LIN {X 0,Y 573.289,Z 87.196,A -85,B 0,C 180,E1 -2345.628,E2 -2345.628} C_VEL
LIN {X 0,Y 573.282,Z 87.197,A -85,B 0,C 180,E1 -2348.46,E2 -2348.46} C_VEL
LIN {X 0,Y 573.272,Z 87.197,A -85,B 0,C 180,E1 -2351.312,E2 -2351.312} C_VEL
LIN {X 0,Y 573.282,Z 87.196,A -85,B 0,C 180,E1 -2354.425,E2 -2354.425} C_VEL
LIN {X 0,Y 573.257,Z 87.199,A -85,B 0,C 180,E1 -2357.112,E2 -2357.112} C_VEL
LIN {X 0,Y 573.248,Z 87.201,A -85,B 0,C 180,E1 -2360.077,E2 -2360.077} C_VEL
LIN {X 0,Y 573.234,Z 87.203,A -85,B 0,C 180,E1 -2363.1,E2 -2363.1} C_VEL
LIN {X 0,Y 573.246,Z 87.199,A -85,B 0,C 180,E1 -2364.375,E2 -2364.375} C_VEL
LIN {X 0,Y 572.621,Z 87.279,A -85,B 0,C 180,E1 -2364.961,E2 -2364.961} C_VEL
LIN {X 0,Y 569.781,Z 87.64,A -85,B 0,C 180,E1 -2365.912,E2 -2365.912} C_VEL
LIN {X 0,Y 567.349,Z 87.946,A -85,B 0,C 180,E1 -2366.678,E2 -2366.678} C_VEL
LIN {X 0,Y 566.294,Z 88.074,A -85,B 0,C 180,E1 -2367.269,E2 -2367.269} C_VEL
LIN {X 0,Y 566.203,Z 88.082,A -85,B 0,C 180,E1 -2367.469,E2 -2367.469} C_VEL
LIN {X 0,Y 566.196,Z 88.08,A -85,B 0,C 180,E1 -2369.769,E2 -2369.769} C_VEL
LIN {X 0,Y 566.202,Z 88.076,A -85,B 0,C 180,E1 -2372.43,E2 -2372.43} C_VEL
LIN {X 0,Y 566.179,Z 88.086,A -85,B 0,C 180,E1 -2374.99,E2 -2374.99} C_VEL
LIN {X 0,Y 566.196,Z 88.08,A -85,B 0,C 180,E1 -2377.461,E2 -2377.461} C_VEL
LIN {X 0,Y 566.207,Z 88.076,A -85,B 0,C 180,E1 -2380.199,E2 -2380.199} C_VEL
LIN {X 0,Y 566.198,Z 88.083,A -85,B 0,C 180,E1 -2383.055,E2 -2383.055} C_VEL
LIN {X 0,Y 566.194,Z 88.078,A -85,B 0,C 180,E1 -2386.05,E2 -2386.05} C_VEL
LIN {X 0,Y 566.204,Z 88.078,A -85,B 0,C 180,E1 -2389.215,E2 -2389.215} C_VEL
LIN {X 0,Y 566.182,Z 88.078,A -85,B 0,C 180,E1 -2391.637,E2 -2391.637} C_VEL
LIN {X 0,Y 566.151,Z 88.089,A -85,B 0,C 180,E1 -2394.307,E2 -2394.307} C_VEL
LIN {X 0,Y 566.221,Z 88.076,A -85,B 0,C 180,E1 -2396.898,E2 -2396.898} C_VEL
LIN {X 0,Y 566.18,Z 88.079,A -85,B 0,C 180,E1 -2399.407,E2 -2399.407} C_VEL
LIN {X 0,Y 566.189,Z 88.081,A -85,B 0,C 180,E1 -2401.856,E2 -2401.856} C_VEL
LIN {X 0,Y 566.24,Z 88.071,A -85,B 0,C 180,E1 -2405.039,E2 -2405.039} C_VEL
LIN {X 0,Y 566.194,Z 88.086,A -85,B 0,C 180,E1 -2408.138,E2 -2408.138} C_VEL
LIN {X 0,Y 566.234,Z 88.075,A -85,B 0,C 180,E1 -2410.614,E2 -2410.614} C_VEL
LIN {X 0,Y 566.2,Z 88.087,A -85,B 0,C 180,E1 -2413.783,E2 -2413.783} C_VEL
LIN {X 0,Y 566.208,Z 88.167,A -85,B 0,C 180,E1 -2414.153,E2 -2414.153} C_VEL
LIN {X 0,Y 566.918,Z 92.77,A -85,B 0,C 180,E1 -2414.91,E2 -2414.91} C_VEL
LIN {X 0,Y 566.626,Z 111.554,A -85,B 0,C 180,E1 -2417.828,E2 -2417.828} C_VEL
LIN {X 0,Y 566.562,Z 119.682,A -85,B 0,C 180,E1 -2419.076,E2 -2419.076} C_VEL
LIN {X 0,Y 567.768,Z 127.51,A -85,B 0,C 180,E1 -2419.22,E2 -2419.22} C_VEL
LIN {X 0,Y 567.41,Z 256.467,A -85,B 0,C 180,E1 -2420.891,E2 -2420.891} C_VEL
LIN {X 0,Y 567.294,Z 270.884,A -85,B 0,C 180,E1 -2421.226,E2 -2421.226} C_VEL
LIN {X 0,Y 567.151,Z 285.238,A -85,B 0,C 180,E1 -2421.718,E2 -2421.718} C_VEL
LIN {X 0,Y 566.971,Z 298.855,A -85,B 0,C 180,E1 -2422.343,E2 -2422.343} C_VEL
LIN {X 0,Y 566.759,Z 311.074,A -85,B 0,C 180,E1 -2423.055,E2 -2423.055} C_VEL
LIN {X 0,Y 566.617,Z 323.455,A -85,B 0,C 180,E1 -2423.948,E2 -2423.948} C_VEL
LIN {X 0,Y 566.381,Z 333.622,A -85,B 0,C 180,E1 -2424.839,E2 -2424.839} C_VEL
LIN {X 0,Y 566.246,Z 343.77,A -85,B 0,C 180,E1 -2425.908,E2 -2425.908} C_VEL
LIN {X 0,Y 566.124,Z 352.189,A -85,B 0,C 180,E1 -2426.976,E2 -2426.976} C_VEL
LIN {X 0,Y 566.109,Z 360.261,A -85,B 0,C 180,E1 -2428.222,E2 -2428.222} C_VEL
LIN {X 0,Y 565.936,Z 365.957,A -85,B 0,C 180,E1 -2429.289,E2 -2429.289} C_VEL
LIN {X 0,Y 565.95,Z 370.617,A -85,B 0,C 180,E1 -2430.356,E2 -2430.356} C_VEL
LIN {X 0,Y 565.9,Z 375.469,A -85,B 0,C 180,E1 -2431.779,E2 -2431.779} C_VEL
LIN {X 0,Y 565.873,Z 378.126,A -85,B 0,C 180,E1 -2432.848,E2 -2432.848} C_VEL
LIN {X 0,Y 565.91,Z 380.449,A -85,B 0,C 180,E1 -2434.273,E2 -2434.273} C_VEL
LIN {X 0,Y 565.895,Z 381.431,A -85,B 0,C 180,E1 -2435.702,E2 -2435.702} C_VEL
LIN {X 0,Y 565.885,Z 381.084,A -85,B 0,C 180,E1 -2437.134,E2 -2437.134} C_VEL
LIN {X 0,Y 565.853,Z 379.389,A -85,B 0,C 180,E1 -2438.572,E2 -2438.572} C_VEL
LIN {X 0,Y 565.913,Z 376.297,A -85,B 0,C 180,E1 -2440.013,E2 -2440.013} C_VEL
LIN {X 0,Y 565.942,Z 371.702,A -85,B 0,C 180,E1 -2441.461,E2 -2441.461} C_VEL
LIN {X 0,Y 565.955,Z 367.124,A -85,B 0,C 180,E1 -2442.551,E2 -2442.551} C_VEL
LIN {X 0,Y 566.033,Z 360.492,A -85,B 0,C 180,E1 -2443.828,E2 -2443.828} C_VEL
LIN {X 0,Y 566.123,Z 352.208,A -85,B 0,C 180,E1 -2445.112,E2 -2445.112} C_VEL
LIN {X 0,Y 566.243,Z 343.476,A -85,B 0,C 180,E1 -2446.216,E2 -2446.216} C_VEL
LIN {X 0,Y 566.418,Z 332.825,A -85,B 0,C 180,E1 -2447.325,E2 -2447.325} C_VEL
LIN {X 0,Y 566.578,Z 322.04,A -85,B 0,C 180,E1 -2448.253,E2 -2448.253} C_VEL
LIN {X 0,Y 566.775,Z 310.231,A -85,B 0,C 180,E1 -2449.089,E2 -2449.089} C_VEL
LIN {X 0,Y 566.988,Z 297.689,A -85,B 0,C 180,E1 -2449.807,E2 -2449.807} C_VEL
LIN {X 0,Y 567.161,Z 284.65,A -85,B 0,C 180,E1 -2450.396,E2 -2450.396} C_VEL
LIN {X 0,Y 567.302,Z 270.052,A -85,B 0,C 180,E1 -2450.889,E2 -2450.889} C_VEL
LIN {X 0,Y 567.409,Z 255.45,A -85,B 0,C 180,E1 -2451.216,E2 -2451.216} C_VEL
LIN {X 0,Y 567.666,Z 125.494,A -85,B 0,C 180,E1 -2452.9,E2 -2452.9} C_VEL
LIN {X 0,Y 566.565,Z 119.617,A -85,B 0,C 180,E1 -2453.025,E2 -2453.025} C_VEL
LIN {X 0,Y 566.783,Z 100.873,A -85,B 0,C 180,E1 -2455.919,E2 -2455.919} C_VEL
LIN {X 0,Y 566.816,Z 92.019,A -85,B 0,C 180,E1 -2457.308,E2 -2457.308} C_VEL
LIN {X 0,Y 566.144,Z 88.093,A -85,B 0,C 180,E1 -2457.995,E2 -2457.995} C_VEL
LIN {X 0,Y 566.173,Z 88.082,A -85,B 0,C 180,E1 -2461.073,E2 -2461.073} C_VEL
LIN {X 0,Y 566.18,Z 88.085,A -85,B 0,C 180,E1 -2463.729,E2 -2463.729} C_VEL
LIN {X 0,Y 566.14,Z 88.085,A -85,B 0,C 180,E1 -2466.574,E2 -2466.574} C_VEL
LIN {X 0,Y 566.194,Z 88.08,A -85,B 0,C 180,E1 -2469.275,E2 -2469.275} C_VEL
LIN {X 0,Y 566.141,Z 88.088,A -85,B 0,C 180,E1 -2472.094,E2 -2472.094} C_VEL
LIN {X 0,Y 566.159,Z 88.084,A -85,B 0,C 180,E1 -2475.037,E2 -2475.037} C_VEL
LIN {X 0,Y 566.15,Z 88.086,A -85,B 0,C 180,E1 -2477.906,E2 -2477.906} C_VEL
LIN {X 0,Y 566.205,Z 88.075,A -85,B 0,C 180,E1 -2480.725,E2 -2480.725} C_VEL
LIN {X 0,Y 566.176,Z 88.086,A -85,B 0,C 180,E1 -2483.428,E2 -2483.428} C_VEL
LIN {X 0,Y 566.197,Z 88.077,A -85,B 0,C 180,E1 -2486.268,E2 -2486.268} C_VEL
LIN {X 0,Y 566.182,Z 88.086,A -85,B 0,C 180,E1 -2488.925,E2 -2488.925} C_VEL
LIN {X 0,Y 566.171,Z 88.081,A -85,B 0,C 180,E1 -2491.855,E2 -2491.855} C_VEL
LIN {X 0,Y 566.187,Z 88.078,A -85,B 0,C 180,E1 -2494.249,E2 -2494.249} C_VEL
LIN {X 0,Y 566.162,Z 88.082,A -85,B 0,C 180,E1 -2497.368,E2 -2497.368} C_VEL
LIN {X 0,Y 566.202,Z 88.076,A -85,B 0,C 180,E1 -2499.662,E2 -2499.662} C_VEL
LIN {X 0,Y 566.18,Z 88.079,A -85,B 0,C 180,E1 -2501.921,E2 -2501.921} C_VEL
LIN {X 0,Y 566.189,Z 88.082,A -85,B 0,C 180,E1 -2504.152,E2 -2504.152} C_VEL
LIN {X 0,Y 566.173,Z 88.088,A -85,B 0,C 180,E1 -2506.358,E2 -2506.358} C_VEL
LIN {X 0,Y 566.236,Z 88.077,A -85,B 0,C 180,E1 -2508.675,E2 -2508.675} C_VEL
LIN {X 0,Y 566.203,Z 88.075,A -85,B 0,C 180,E1 -2511.434,E2 -2511.434} C_VEL
LIN {X 0,Y 566.255,Z 88.076,A -85,B 0,C 180,E1 -2514.302,E2 -2514.302} C_VEL
LIN {X 0,Y 566.281,Z 88.073,A -85,B 0,C 180,E1 -2517.866,E2 -2517.866} C_VEL
LIN {X 0,Y 566.298,Z 88.063,A -85,B 0,C 180,E1 -2520.711,E2 -2520.711} C_VEL
LIN {X 0,Y 566.267,Z 88.068,A -85,B 0,C 180,E1 -2522.845,E2 -2522.845} C_VEL
LIN {X 0,Y 566.249,Z 88.079,A -85,B 0,C 180,E1 -2525.698,E2 -2525.698} C_VEL
LIN {X 0,Y 566.225,Z 88.074,A -85,B 0,C 180,E1 -2528.566,E2 -2528.566} C_VEL
LIN {X 0,Y 566.243,Z 88.079,A -85,B 0,C 180,E1 -2531.454,E2 -2531.454} C_VEL
LIN {X 0,Y 566.224,Z 88.074,A -85,B 0,C 180,E1 -2534.502,E2 -2534.502} C_VEL
LIN {X 0,Y 566.2,Z 88.085,A -85,B 0,C 180,E1 -2537.332,E2 -2537.332} C_VEL
LIN {X 0,Y 566.207,Z 88.075,A -85,B 0,C 180,E1 -2540.337,E2 -2540.337} C_VEL
LIN {X 0,Y 566.17,Z 88.086,A -85,B 0,C 180,E1 -2543.281,E2 -2543.281} C_VEL
LIN {X 0,Y 566.216,Z 88.075,A -85,B 0,C 180,E1 -2545.749,E2 -2545.749} C_VEL
LIN {X 0,Y 566.204,Z 88.076,A -85,B 0,C 180,E1 -2548.202,E2 -2548.202} C_VEL
LIN {X 0,Y 566.199,Z 88.081,A -85,B 0,C 180,E1 -2551.078,E2 -2551.078} C_VEL
LIN {X 0,Y 566.213,Z 88.075,A -85,B 0,C 180,E1 -2553.734,E2 -2553.734} C_VEL
LIN {X 0,Y 566.2,Z 88.085,A -85,B 0,C 180,E1 -2556.57,E2 -2556.57} C_VEL
LIN {X 0,Y 566.216,Z 88.072,A -85,B 0,C 180,E1 -2559.686,E2 -2559.686} C_VEL
LIN {X 0,Y 566.212,Z 88.08,A -85,B 0,C 180,E1 -2562.087,E2 -2562.087} C_VEL
LIN {X 0,Y 566.169,Z 88.08,A -85,B 0,C 180,E1 -2565.036,E2 -2565.036} C_VEL
LIN {X 0,Y 566.19,Z 88.083,A -85,B 0,C 180,E1 -2567.91,E2 -2567.91} C_VEL
LIN {X 0,Y 566.223,Z 88.074,A -85,B 0,C 180,E1 -2570.727,E2 -2570.727} C_VEL
LIN {X 0,Y 566.186,Z 88.085,A -85,B 0,C 180,E1 -2573.788,E2 -2573.788} C_VEL
LIN {X 0,Y 566.213,Z 88.077,A -85,B 0,C 180,E1 -2576.266,E2 -2576.266} C_VEL
LIN {X 0,Y 566.192,Z 88.078,A -85,B 0,C 180,E1 -2578.924,E2 -2578.924} C_VEL
LIN {X 0,Y 566.213,Z 88.083,A -85,B 0,C 180,E1 -2581.857,E2 -2581.857} C_VEL
LIN {X 0,Y 566.214,Z 88.079,A -85,B 0,C 180,E1 -2584.251,E2 -2584.251} C_VEL
LIN {X 0,Y 566.257,Z 88.279,A -85,B 0,C 180,E1 -2585.529,E2 -2585.529} C_VEL
LIN {X 0,Y 567.225,Z 92.989,A -85,B 0,C 180,E1 -2586.223,E2 -2586.223} C_VEL
LIN {X 0,Y 567.081,Z 109.533,A -85,B 0,C 180,E1 -2588.477,E2 -2588.477} C_VEL
LIN {X 0,Y 566.824,Z 129.821,A -85,B 0,C 180,E1 -2591.194,E2 -2591.194} C_VEL
LIN {X 0,Y 566.669,Z 143.602,A -85,B 0,C 180,E1 -2593.018,E2 -2593.018} C_VEL
LIN {X 0,Y 567.796,Z 150.524,A -85,B 0,C 180,E1 -2593.151,E2 -2593.151} C_VEL
LIN {X 0,Y 567.401,Z 281.88,A -85,B 0,C 180,E1 -2594.854,E2 -2594.854} C_VEL
LIN {X 0,Y 567.27,Z 296.576,A -85,B 0,C 180,E1 -2595.201,E2 -2595.201} C_VEL
LIN {X 0,Y 567.111,Z 310.832,A -85,B 0,C 180,E1 -2595.695,E2 -2595.695} C_VEL
LIN {X 0,Y 566.966,Z 323.636,A -85,B 0,C 180,E1 -2596.286,E2 -2596.286} C_VEL
LIN {X 0,Y 566.787,Z 336.098,A -85,B 0,C 180,E1 -2597.012,E2 -2597.012} C_VEL
LIN {X 0,Y 566.578,Z 347.481,A -85,B 0,C 180,E1 -2597.826,E2 -2597.826} C_VEL
LIN {X 0,Y 566.412,Z 358.006,A -85,B 0,C 180,E1 -2598.737,E2 -2598.737} C_VEL
LIN {X 0,Y 566.247,Z 368.332,A -85,B 0,C 180,E1 -2599.813,E2 -2599.813} C_VEL
LIN {X 0,Y 566.152,Z 376.91,A -85,B 0,C 180,E1 -2600.893,E2 -2600.893} C_VEL
LIN {X 0,Y 566.059,Z 385.117,A -85,B 0,C 180,E1 -2602.15,E2 -2602.15} C_VEL
LIN {X 0,Y 565.966,Z 391.802,A -85,B 0,C 180,E1 -2603.422,E2 -2603.422} C_VEL
LIN {X 0,Y 565.927,Z 396.96,A -85,B 0,C 180,E1 -2604.656,E2 -2604.656} C_VEL
LIN {X 0,Y 565.957,Z 400.443,A -85,B 0,C 180,E1 -2605.727,E2 -2605.727} C_VEL
LIN {X 0,Y 565.874,Z 403.832,A -85,B 0,C 180,E1 -2607.152,E2 -2607.152} C_VEL
LIN {X 0,Y 565.841,Z 405.834,A -85,B 0,C 180,E1 -2608.576,E2 -2608.576} C_VEL
LIN {X 0,Y 565.837,Z 406.5,A -85,B 0,C 180,E1 -2610,E2 -2610} C_VEL
LIN {X 0,Y 565.841,Z 405.835,A -85,B 0,C 180,E1 -2611.423,E2 -2611.423} C_VEL
LIN {X 0,Y 565.874,Z 403.835,A -85,B 0,C 180,E1 -2612.847,E2 -2612.847} C_VEL
LIN {X 0,Y 565.957,Z 400.447,A -85,B 0,C 180,E1 -2614.273,E2 -2614.273} C_VEL
LIN {X 0,Y 565.985,Z 395.568,A -85,B 0,C 180,E1 -2615.701,E2 -2615.701} C_VEL
LIN {X 0,Y 565.995,Z 391.044,A -85,B 0,C 180,E1 -2616.739,E2 -2616.739} C_VEL
LIN {X 0,Y 566.047,Z 384.036,A -85,B 0,C 180,E1 -2618.029,E2 -2618.029} C_VEL
LIN {X 0,Y 566.177,Z 375.558,A -85,B 0,C 180,E1 -2619.286,E2 -2619.286} C_VEL
LIN {X 0,Y 566.294,Z 366.708,A -85,B 0,C 180,E1 -2620.367,E2 -2620.367} C_VEL
LIN {X 0,Y 566.485,Z 355.988,A -85,B 0,C 180,E1 -2621.449,E2 -2621.449} C_VEL
LIN {X 0,Y 566.611,Z 345.137,A -85,B 0,C 180,E1 -2622.354,E2 -2622.354} C_VEL
LIN {X 0,Y 566.8,Z 333.254,A -85,B 0,C 180,E1 -2623.17,E2 -2623.17} C_VEL
LIN {X 0,Y 567.009,Z 320.098,A -85,B 0,C 180,E1 -2623.895,E2 -2623.895} C_VEL
LIN {X 0,Y 567.242,Z 307.058,A -85,B 0,C 180,E1 -2624.452,E2 -2624.452} C_VEL
LIN {X 0,Y 567.324,Z 293.236,A -85,B 0,C 180,E1 -2624.892,E2 -2624.892} C_VEL
LIN {X 0,Y 567.449,Z 279.137,A -85,B 0,C 180,E1 -2625.19,E2 -2625.19} C_VEL
LIN {X 0,Y 567.732,Z 149.651,A -85,B 0,C 180,E1 -2626.863,E2 -2626.863} C_VEL
LIN {X 0,Y 566.664,Z 143.605,A -85,B 0,C 180,E1 -2626.982,E2 -2626.982} C_VEL
LIN {X 0,Y 566.934,Z 122.933,A -85,B 0,C 180,E1 -2629.724,E2 -2629.724} C_VEL
LIN {X 0,Y 567.203,Z 101.667,A -85,B 0,C 180,E1 -2632.588,E2 -2632.588} C_VEL
LIN {X 0,Y 567.225,Z 92.993,A -85,B 0,C 180,E1 -2633.779,E2 -2633.779} C_VEL
LIN {X 0,Y 566.241,Z 88.08,A -85,B 0,C 180,E1 -2634.52,E2 -2634.52} C_VEL
LIN {X 0,Y 566.212,Z 88.076,A -85,B 0,C 180,E1 -2637.339,E2 -2637.339} C_VEL
LIN {X 0,Y 566.201,Z 88.08,A -85,B 0,C 180,E1 -2639.769,E2 -2639.769} C_VEL
LIN {X 0,Y 566.204,Z 88.082,A -85,B 0,C 180,E1 -2642.43,E2 -2642.43} C_VEL
LIN {X 0,Y 566.181,Z 88.079,A -85,B 0,C 180,E1 -2644.989,E2 -2644.989} C_VEL
LIN {X 0,Y 566.197,Z 88.078,A -85,B 0,C 180,E1 -2647.461,E2 -2647.461} C_VEL
LIN {X 0,Y 566.218,Z 88.08,A -85,B 0,C 180,E1 -2650.198,E2 -2650.198} C_VEL
LIN {X 0,Y 566.201,Z 88.077,A -85,B 0,C 180,E1 -2653.054,E2 -2653.054} C_VEL
LIN {X 0,Y 566.202,Z 88.081,A -85,B 0,C 180,E1 -2656.048,E2 -2656.048} C_VEL
LIN {X 0,Y 566.182,Z 88.079,A -85,B 0,C 180,E1 -2658.861,E2 -2658.861} C_VEL
LIN {X 0,Y 566.185,Z 88.087,A -85,B 0,C 180,E1 -2661.637,E2 -2661.637} C_VEL
LIN {X 0,Y 566.162,Z 88.081,A -85,B 0,C 180,E1 -2664.308,E2 -2664.308} C_VEL
LIN {X 0,Y 566.228,Z 88.075,A -85,B 0,C 180,E1 -2666.898,E2 -2666.898} C_VEL
LIN {X 0,Y 566.184,Z 88.087,A -85,B 0,C 180,E1 -2669.407,E2 -2669.407} C_VEL
LIN {X 0,Y 566.211,Z 88.076,A -85,B 0,C 180,E1 -2671.857,E2 -2671.857} C_VEL
LIN {X 0,Y 566.214,Z 88.075,A -85,B 0,C 180,E1 -2674.251,E2 -2674.251} C_VEL
LIN {X 0,Y 566.172,Z 88.084,A -85,B 0,C 180,E1 -2676.718,E2 -2676.718} C_VEL
LIN {X 0,Y 566.206,Z 88.076,A -85,B 0,C 180,E1 -2679.663,E2 -2679.663} C_VEL
LIN {X 0,Y 566.198,Z 88.083,A -85,B 0,C 180,E1 -2682.668,E2 -2682.668} C_VEL
LIN {X 0,Y 566.234,Z 88.072,A -85,B 0,C 180,E1 -2685.627,E2 -2685.627} C_VEL
LIN {X 0,Y 566.234,Z 88.082,A -85,B 0,C 180,E1 -2688.675,E2 -2688.675} C_VEL
LIN {X 0,Y 566.227,Z 88.073,A -85,B 0,C 180,E1 -2691.434,E2 -2691.434} C_VEL
LIN {X 0,Y 566.255,Z 88.076,A -85,B 0,C 180,E1 -2694.302,E2 -2694.302} C_VEL
LIN {X 0,Y 566.279,Z 88.069,A -85,B 0,C 180,E1 -2697.866,E2 -2697.866} C_VEL
LIN {X 0,Y 566.299,Z 88.067,A -85,B 0,C 180,E1 -2700.711,E2 -2700.711} C_VEL
LIN {X 0,Y 566.268,Z 88.069,A -85,B 0,C 180,E1 -2702.846,E2 -2702.846} C_VEL
LIN {X 0,Y 566.255,Z 88.073,A -85,B 0,C 180,E1 -2705.698,E2 -2705.698} C_VEL
LIN {X 0,Y 566.227,Z 88.075,A -85,B 0,C 180,E1 -2708.566,E2 -2708.566} C_VEL
LIN {X 0,Y 566.242,Z 88.074,A -85,B 0,C 180,E1 -2711.454,E2 -2711.454} C_VEL
LIN {X 0,Y 566.235,Z 88.073,A -85,B 0,C 180,E1 -2714.507,E2 -2714.507} C_VEL
LIN {X 0,Y 566.196,Z 88.08,A -85,B 0,C 180,E1 -2717.332,E2 -2717.332} C_VEL
LIN {X 0,Y 566.211,Z 88.076,A -85,B 0,C 180,E1 -2720.337,E2 -2720.337} C_VEL
LIN {X 0,Y 566.171,Z 88.085,A -85,B 0,C 180,E1 -2723.282,E2 -2723.282} C_VEL
LIN {X 0,Y 566.21,Z 88.08,A -85,B 0,C 180,E1 -2725.749,E2 -2725.749} C_VEL
LIN {X 0,Y 566.203,Z 88.082,A -85,B 0,C 180,E1 -2727.469,E2 -2727.469} C_VEL
LIN {X 0,Y 565.522,Z 88.163,A -85,B 0,C 180,E1 -2728.063,E2 -2728.063} C_VEL
LIN {X 0,Y 562.655,Z 88.523,A -85,B 0,C 180,E1 -2729.026,E2 -2729.026} C_VEL
LIN {X 0,Y 560.243,Z 88.821,A -85,B 0,C 180,E1 -2729.802,E2 -2729.802} C_VEL
LIN {X 0,Y 559.215,Z 88.947,A -85,B 0,C 180,E1 -2730.401,E2 -2730.401} C_VEL
LIN {X 0,Y 559.134,Z 88.957,A -85,B 0,C 180,E1 -2730.603,E2 -2730.603} C_VEL
LIN {X 0,Y 559.152,Z 88.957,A -85,B 0,C 180,E1 -2732.716,E2 -2732.716} C_VEL
LIN {X 0,Y 559.127,Z 88.964,A -85,B 0,C 180,E1 -2735.324,E2 -2735.324} C_VEL
LIN {X 0,Y 559.131,Z 88.957,A -85,B 0,C 180,E1 -2738.018,E2 -2738.018} C_VEL
LIN {X 0,Y 559.155,Z 88.961,A -85,B 0,C 180,E1 -2740.813,E2 -2740.813} C_VEL
LIN {X 0,Y 559.138,Z 88.956,A -85,B 0,C 180,E1 -2743.735,E2 -2743.735} C_VEL
LIN {X 0,Y 559.143,Z 88.965,A -85,B 0,C 180,E1 -2746.804,E2 -2746.804} C_VEL
LIN {X 0,Y 559.156,Z 88.956,A -85,B 0,C 180,E1 -2749.188,E2 -2749.188} C_VEL
LIN {X 0,Y 559.13,Z 88.959,A -85,B 0,C 180,E1 -2751.982,E2 -2751.982} C_VEL
LIN {X 0,Y 559.129,Z 88.962,A -85,B 0,C 180,E1 -2754.788,E2 -2754.788} C_VEL
LIN {X 0,Y 559.157,Z 88.954,A -85,B 0,C 180,E1 -2757.365,E2 -2757.365} C_VEL
LIN {X 0,Y 559.149,Z 88.961,A -85,B 0,C 180,E1 -2760.143,E2 -2760.143} C_VEL
LIN {X 0,Y 559.121,Z 88.958,A -85,B 0,C 180,E1 -2763.183,E2 -2763.183} C_VEL
LIN {X 0,Y 559.157,Z 88.955,A -85,B 0,C 180,E1 -2765.495,E2 -2765.495} C_VEL
LIN {X 0,Y 559.174,Z 88.954,A -85,B 0,C 180,E1 -2768.624,E2 -2768.624} C_VEL
LIN {X 0,Y 559.163,Z 88.955,A -85,B 0,C 180,E1 -2770.926,E2 -2770.926} C_VEL
LIN {X 0,Y 559.166,Z 88.963,A -85,B 0,C 180,E1 -2773.948,E2 -2773.948} C_VEL
LIN {X 0,Y 559.976,Z 93.437,A -85,B 0,C 180,E1 -2774.719,E2 -2774.719} C_VEL
LIN {X 0,Y 559.692,Z 112.222,A -85,B 0,C 180,E1 -2777.675,E2 -2777.675} C_VEL
LIN {X 0,Y 559.619,Z 119.863,A -85,B 0,C 180,E1 -2778.863,E2 -2778.863} C_VEL
LIN {X 0,Y 560.969,Z 128.465,A -85,B 0,C 180,E1 -2779.02,E2 -2779.02} C_VEL
LIN {X 0,Y 560.574,Z 257.017,A -85,B 0,C 180,E1 -2780.711,E2 -2780.711} C_VEL
LIN {X 0,Y 560.443,Z 271.272,A -85,B 0,C 180,E1 -2781.05,E2 -2781.05} C_VEL
LIN {X 0,Y 560.295,Z 284.973,A -85,B 0,C 180,E1 -2781.525,E2 -2781.525} C_VEL
LIN {X 0,Y 560.078,Z 298.637,A -85,B 0,C 180,E1 -2782.157,E2 -2782.157} C_VEL
LIN {X 0,Y 559.829,Z 310.765,A -85,B 0,C 180,E1 -2782.87,E2 -2782.87} C_VEL
LIN {X 0,Y 559.656,Z 322.136,A -85,B 0,C 180,E1 -2783.692,E2 -2783.692} C_VEL
LIN {X 0,Y 559.419,Z 332.519,A -85,B 0,C 180,E1 -2784.594,E2 -2784.594} C_VEL
LIN {X 0,Y 559.199,Z 342.866,A -85,B 0,C 180,E1 -2785.675,E2 -2785.675} C_VEL
LIN {X 0,Y 559.107,Z 351.426,A -85,B 0,C 180,E1 -2786.757,E2 -2786.757} C_VEL
LIN {X 0,Y 558.962,Z 359.679,A -85,B 0,C 180,E1 -2788.019,E2 -2788.019} C_VEL
LIN {X 0,Y 558.847,Z 366.334,A -85,B 0,C 180,E1 -2789.28,E2 -2789.28} C_VEL
LIN {X 0,Y 558.793,Z 372.263,A -85,B 0,C 180,E1 -2790.721,E2 -2790.721} C_VEL
LIN {X 0,Y 558.747,Z 376.637,A -85,B 0,C 180,E1 -2792.163,E2 -2792.163} C_VEL
LIN {X 0,Y 558.818,Z 379.575,A -85,B 0,C 180,E1 -2793.605,E2 -2793.605} C_VEL
LIN {X 0,Y 558.76,Z 381.156,A -85,B 0,C 180,E1 -2795.051,E2 -2795.051} C_VEL
LIN {X 0,Y 558.847,Z 381.398,A -85,B 0,C 180,E1 -2796.536,E2 -2796.536} C_VEL
LIN {X 0,Y 558.796,Z 380.32,A -85,B 0,C 180,E1 -2797.952,E2 -2797.952} C_VEL
LIN {X 0,Y 558.751,Z 377.864,A -85,B 0,C 180,E1 -2799.411,E2 -2799.411} C_VEL
LIN {X 0,Y 558.855,Z 373.958,A -85,B 0,C 180,E1 -2800.873,E2 -2800.873} C_VEL
LIN {X 0,Y 558.848,Z 369.952,A -85,B 0,C 180,E1 -2801.976,E2 -2801.976} C_VEL
LIN {X 0,Y 558.898,Z 364.985,A -85,B 0,C 180,E1 -2803.082,E2 -2803.082} C_VEL
LIN {X 0,Y 559.025,Z 357.558,A -85,B 0,C 180,E1 -2804.417,E2 -2804.417} C_VEL
LIN {X 0,Y 559.142,Z 348.856,A -85,B 0,C 180,E1 -2805.679,E2 -2805.679} C_VEL
LIN {X 0,Y 559.302,Z 339.434,A -85,B 0,C 180,E1 -2806.799,E2 -2806.799} C_VEL
LIN {X 0,Y 559.501,Z 328.945,A -85,B 0,C 180,E1 -2807.829,E2 -2807.829} C_VEL
LIN {X 0,Y 559.722,Z 317.287,A -85,B 0,C 180,E1 -2808.769,E2 -2808.769} C_VEL
LIN {X 0,Y 559.937,Z 304.599,A -85,B 0,C 180,E1 -2809.602,E2 -2809.602} C_VEL
LIN {X 0,Y 560.158,Z 291.637,A -85,B 0,C 180,E1 -2810.279,E2 -2810.279} C_VEL
LIN {X 0,Y 560.379,Z 278.781,A -85,B 0,C 180,E1 -2810.799,E2 -2810.799} C_VEL
LIN {X 0,Y 560.484,Z 265.183,A -85,B 0,C 180,E1 -2811.203,E2 -2811.203} C_VEL
LIN {X 0,Y 560.6,Z 251.707,A -85,B 0,C 180,E1 -2811.465,E2 -2811.465} C_VEL
LIN {X 0,Y 560.981,Z 126.863,A -85,B 0,C 180,E1 -2813.09,E2 -2813.09} C_VEL
LIN {X 0,Y 559.588,Z 119.741,A -85,B 0,C 180,E1 -2813.249,E2 -2813.249} C_VEL
LIN {X 0,Y 559.854,Z 101.738,A -85,B 0,C 180,E1 -2816.063,E2 -2816.063} C_VEL
LIN {X 0,Y 559.843,Z 92.938,A -85,B 0,C 180,E1 -2817.462,E2 -2817.462} C_VEL
LIN {X 0,Y 559.088,Z 88.972,A -85,B 0,C 180,E1 -2818.157,E2 -2818.157} C_VEL
LIN {X 0,Y 559.138,Z 88.959,A -85,B 0,C 180,E1 -2821.02,E2 -2821.02} C_VEL
LIN {X 0,Y 559.141,Z 88.965,A -85,B 0,C 180,E1 -2823.945,E2 -2823.945} C_VEL
LIN {X 0,Y 559.11,Z 88.96,A -85,B 0,C 180,E1 -2827.111,E2 -2827.111} C_VEL
LIN {X 0,Y 559.121,Z 88.966,A -85,B 0,C 180,E1 -2829.936,E2 -2829.936} C_VEL
LIN {X 0,Y 559.108,Z 88.96,A -85,B 0,C 180,E1 -2832.748,E2 -2832.748} C_VEL
LIN {X 0,Y 559.122,Z 88.964,A -85,B 0,C 180,E1 -2835.764,E2 -2835.764} C_VEL
LIN {X 0,Y 559.102,Z 88.962,A -85,B 0,C 180,E1 -2838.224,E2 -2838.224} C_VEL
LIN {X 0,Y 559.168,Z 88.954,A -85,B 0,C 180,E1 -2841.065,E2 -2841.065} C_VEL
LIN {X 0,Y 559.117,Z 88.961,A -85,B 0,C 180,E1 -2843.787,E2 -2843.787} C_VEL
LIN {X 0,Y 559.146,Z 88.956,A -85,B 0,C 180,E1 -2846.424,E2 -2846.424} C_VEL
LIN {X 0,Y 559.146,Z 88.963,A -85,B 0,C 180,E1 -2848.98,E2 -2848.98} C_VEL
LIN {X 0,Y 559.114,Z 88.961,A -85,B 0,C 180,E1 -2851.629,E2 -2851.629} C_VEL
LIN {X 0,Y 559.155,Z 88.953,A -85,B 0,C 180,E1 -2853.901,E2 -2853.901} C_VEL
LIN {X 0,Y 559.112,Z 88.963,A -85,B 0,C 180,E1 -2857.066,E2 -2857.066} C_VEL
LIN {X 0,Y 559.173,Z 88.953,A -85,B 0,C 180,E1 -2859.395,E2 -2859.395} C_VEL
LIN {X 0,Y 559.129,Z 88.956,A -85,B 0,C 180,E1 -2861.685,E2 -2861.685} C_VEL
LIN {X 0,Y 559.153,Z 88.956,A -85,B 0,C 180,E1 -2863.947,E2 -2863.947} C_VEL
LIN {X 0,Y 559.15,Z 88.957,A -85,B 0,C 180,E1 -2866.924,E2 -2866.924} C_VEL
LIN {X 0,Y 559.191,Z 88.95,A -85,B 0,C 180,E1 -2869.133,E2 -2869.133} C_VEL
LIN {X 0,Y 559.195,Z 88.954,A -85,B 0,C 180,E1 -2872.053,E2 -2872.053} C_VEL
LIN {X 0,Y 559.244,Z 88.943,A -85,B 0,C 180,E1 -2874.953,E2 -2874.953} C_VEL
LIN {X 0,Y 559.252,Z 88.948,A -85,B 0,C 180,E1 -2877.839,E2 -2877.839} C_VEL
LIN {X 0,Y 559.269,Z 88.939,A -85,B 0,C 180,E1 -2880.72,E2 -2880.72} C_VEL
LIN {X 0,Y 559.233,Z 88.944,A -85,B 0,C 180,E1 -2882.881,E2 -2882.881} C_VEL
LIN {X 0,Y 559.218,Z 88.953,A -85,B 0,C 180,E1 -2885.77,E2 -2885.77} C_VEL
LIN {X 0,Y 559.184,Z 88.951,A -85,B 0,C 180,E1 -2888.674,E2 -2888.674} C_VEL
LIN {X 0,Y 559.206,Z 88.955,A -85,B 0,C 180,E1 -2891.6,E2 -2891.6} C_VEL
LIN {X 0,Y 559.181,Z 88.951,A -85,B 0,C 180,E1 -2894.587,E2 -2894.587} C_VEL
LIN {X 0,Y 559.159,Z 88.959,A -85,B 0,C 180,E1 -2897.557,E2 -2897.557} C_VEL
LIN {X 0,Y 559.166,Z 88.953,A -85,B 0,C 180,E1 -2899.838,E2 -2899.838} C_VEL
LIN {X 0,Y 559.14,Z 88.955,A -85,B 0,C 180,E1 -2902.153,E2 -2902.153} C_VEL
LIN {X 0,Y 559.177,Z 88.956,A -85,B 0,C 180,E1 -2905.298,E2 -2905.298} C_VEL
LIN {X 0,Y 559.158,Z 88.954,A -85,B 0,C 180,E1 -2907.713,E2 -2907.713} C_VEL
LIN {X 0,Y 559.158,Z 88.955,A -85,B 0,C 180,E1 -2910.182,E2 -2910.182} C_VEL
LIN {X 0,Y 559.176,Z 88.959,A -85,B 0,C 180,E1 -2912.714,E2 -2912.714} C_VEL
LIN {X 0,Y 559.131,Z 88.957,A -85,B 0,C 180,E1 -2915.324,E2 -2915.324} C_VEL
LIN {X 0,Y 559.133,Z 88.959,A -85,B 0,C 180,E1 -2918.018,E2 -2918.018} C_VEL
LIN {X 0,Y 559.159,Z 88.957,A -85,B 0,C 180,E1 -2920.812,E2 -2920.812} C_VEL
LIN {X 0,Y 559.148,Z 88.955,A -85,B 0,C 180,E1 -2923.197,E2 -2923.197} C_VEL
LIN {X 0,Y 559.157,Z 88.963,A -85,B 0,C 180,E1 -2926.268,E2 -2926.268} C_VEL
LIN {X 0,Y 559.175,Z 88.952,A -85,B 0,C 180,E1 -2929.189,E2 -2929.189} C_VEL
LIN {X 0,Y 559.136,Z 88.965,A -85,B 0,C 180,E1 -2931.983,E2 -2931.983} C_VEL
LIN {X 0,Y 559.133,Z 88.957,A -85,B 0,C 180,E1 -2934.787,E2 -2934.787} C_VEL
LIN {X 0,Y 559.157,Z 88.955,A -85,B 0,C 180,E1 -2937.364,E2 -2937.364} C_VEL
LIN {X 0,Y 559.15,Z 88.96,A -85,B 0,C 180,E1 -2940.143,E2 -2940.143} C_VEL
LIN {X 0,Y 559.171,Z 88.956,A -85,B 0,C 180,E1 -2943.098,E2 -2943.098} C_VEL
LIN {X 0,Y 559.234,Z 89.034,A -85,B 0,C 180,E1 -2945.327,E2 -2945.327} C_VEL
LIN {X 0,Y 560.367,Z 95.898,A -85,B 0,C 180,E1 -2946.338,E2 -2946.338} C_VEL
LIN {X 0,Y 560.087,Z 115.602,A -85,B 0,C 180,E1 -2949.046,E2 -2949.046} C_VEL
LIN {X 0,Y 559.807,Z 136.709,A -85,B 0,C 180,E1 -2951.897,E2 -2951.897} C_VEL
LIN {X 0,Y 559.699,Z 143.503,A -85,B 0,C 180,E1 -2952.807,E2 -2952.807} C_VEL
LIN {X 0,Y 560.987,Z 150.895,A -85,B 0,C 180,E1 -2952.947,E2 -2952.947} C_VEL
LIN {X 0,Y 560.561,Z 281.8,A -85,B 0,C 180,E1 -2954.665,E2 -2954.665} C_VEL
LIN {X 0,Y 560.421,Z 296.358,A -85,B 0,C 180,E1 -2955.011,E2 -2955.011} C_VEL
LIN {X 0,Y 560.234,Z 310.8,A -85,B 0,C 180,E1 -2955.516,E2 -2955.516} C_VEL
LIN {X 0,Y 560.067,Z 323.634,A -85,B 0,C 180,E1 -2956.114,E2 -2956.114} C_VEL
LIN {X 0,Y 559.841,Z 336.095,A -85,B 0,C 180,E1 -2956.848,E2 -2956.848} C_VEL
LIN {X 0,Y 559.617,Z 347.478,A -85,B 0,C 180,E1 -2957.673,E2 -2957.673} C_VEL
LIN {X 0,Y 559.388,Z 358.751,A -85,B 0,C 180,E1 -2958.664,E2 -2958.664} C_VEL
LIN {X 0,Y 559.239,Z 368.332,A -85,B 0,C 180,E1 -2959.684,E2 -2959.684} C_VEL
LIN {X 0,Y 559.114,Z 376.909,A -85,B 0,C 180,E1 -2960.778,E2 -2960.778} C_VEL
LIN {X 0,Y 558.98,Z 385.117,A -85,B 0,C 180,E1 -2962.05,E2 -2962.05} C_VEL
LIN {X 0,Y 558.894,Z 392.165,A -85,B 0,C 180,E1 -2963.42,E2 -2963.42} C_VEL
LIN {X 0,Y 558.858,Z 396.96,A -85,B 0,C 180,E1 -2964.588,E2 -2964.588} C_VEL
LIN {X 0,Y 558.866,Z 400.444,A -85,B 0,C 180,E1 -2965.673,E2 -2965.673} C_VEL
LIN {X 0,Y 558.795,Z 403.832,A -85,B 0,C 180,E1 -2967.116,E2 -2967.116} C_VEL
LIN {X 0,Y 558.741,Z 405.834,A -85,B 0,C 180,E1 -2968.558,E2 -2968.558} C_VEL
LIN {X 0,Y 558.738,Z 406.5,A -85,B 0,C 180,E1 -2970,E2 -2970} C_VEL
LIN {X 0,Y 558.741,Z 405.836,A -85,B 0,C 180,E1 -2971.441,E2 -2971.441} C_VEL
LIN {X 0,Y 558.795,Z 403.836,A -85,B 0,C 180,E1 -2972.884,E2 -2972.884} C_VEL
LIN {X 0,Y 558.866,Z 400.447,A -85,B 0,C 180,E1 -2974.327,E2 -2974.327} C_VEL
LIN {X 0,Y 558.914,Z 395.568,A -85,B 0,C 180,E1 -2975.773,E2 -2975.773} C_VEL
LIN {X 0,Y 558.906,Z 389.055,A -85,B 0,C 180,E1 -2977.224,E2 -2977.224} C_VEL
LIN {X 0,Y 559.028,Z 381.804,A -85,B 0,C 180,E1 -2978.495,E2 -2978.495} C_VEL
LIN {X 0,Y 559.146,Z 372.823,A -85,B 0,C 180,E1 -2979.769,E2 -2979.769} C_VEL
LIN {X 0,Y 559.35,Z 363.394,A -85,B 0,C 180,E1 -2980.863,E2 -2980.863} C_VEL
LIN {X 0,Y 559.518,Z 352.953,A -85,B 0,C 180,E1 -2981.869,E2 -2981.869} C_VEL
LIN {X 0,Y 559.696,Z 341.429,A -85,B 0,C 180,E1 -2982.786,E2 -2982.786} C_VEL
LIN {X 0,Y 559.951,Z 328.64,A -85,B 0,C 180,E1 -2983.611,E2 -2983.611} C_VEL
LIN {X 0,Y 560.141,Z 316.127,A -85,B 0,C 180,E1 -2984.254,E2 -2984.254} C_VEL
LIN {X 0,Y 560.384,Z 302.223,A -85,B 0,C 180,E1 -2984.804,E2 -2984.804} C_VEL
LIN {X 0,Y 560.511,Z 288.562,A -85,B 0,C 180,E1 -2985.194,E2 -2985.194} C_VEL
LIN {X 0,Y 560.608,Z 274.525,A -85,B 0,C 180,E1 -2985.45,E2 -2985.45} C_VEL
LIN {X 0,Y 560.965,Z 150.745,A -85,B 0,C 180,E1 -2987.056,E2 -2987.056} C_VEL
LIN {X 0,Y 559.7,Z 143.358,A -85,B 0,C 180,E1 -2987.213,E2 -2987.213} C_VEL
LIN {X 0,Y 560.028,Z 121.241,A -85,B 0,C 180,E1 -2990.188,E2 -2990.188} C_VEL
LIN {X 0,Y 560.416,Z 97.324,A -85,B 0,C 180,E1 -2993.463,E2 -2993.463} C_VEL
LIN {X 0,Y 560.056,Z 93.106,A -85,B 0,C 180,E1 -2994.068,E2 -2994.068} C_VEL
LIN {X 0,Y 559.221,Z 88.955,A -85,B 0,C 180,E1 -2994.698,E2 -2994.698} C_VEL
LIN {X 0,Y 559.182,Z 88.953,A -85,B 0,C 180,E1 -2997.712,E2 -2997.712} C_VEL
LIN {X 0,Y 559.154,Z 88.963,A -85,B 0,C 180,E1 -3000.183,E2 -3000.183} C_VEL
LIN {X 0,Y 559.157,Z 88.956,A -85,B 0,C 180,E1 -3002.715,E2 -3002.715} C_VEL
LIN {X 0,Y 559.128,Z 88.958,A -85,B 0,C 180,E1 -3005.324,E2 -3005.324} C_VEL
LIN {X 0,Y 559.136,Z 88.966,A -85,B 0,C 180,E1 -3008.017,E2 -3008.017} C_VEL
LIN {X 0,Y 559.174,Z 88.952,A -85,B 0,C 180,E1 -3010.811,E2 -3010.811} C_VEL
LIN {X 0,Y 559.141,Z 88.964,A -85,B 0,C 180,E1 -3013.734,E2 -3013.734} C_VEL
LIN {X 0,Y 559.168,Z 88.952,A -85,B 0,C 180,E1 -3016.801,E2 -3016.801} C_VEL
LIN {X 0,Y 559.158,Z 88.956,A -85,B 0,C 180,E1 -3019.188,E2 -3019.188} C_VEL
LIN {X 0,Y 559.132,Z 88.96,A -85,B 0,C 180,E1 -3021.982,E2 -3021.982} C_VEL
LIN {X 0,Y 559.132,Z 88.958,A -85,B 0,C 180,E1 -3024.787,E2 -3024.787} C_VEL
LIN {X 0,Y 559.173,Z 88.961,A -85,B 0,C 180,E1 -3027.361,E2 -3027.361} C_VEL
LIN {X 0,Y 559.148,Z 88.955,A -85,B 0,C 180,E1 -3030.142,E2 -3030.142} C_VEL
LIN {X 0,Y 559.169,Z 88.96,A -85,B 0,C 180,E1 -3033.098,E2 -3033.098} C_VEL
LIN {X 0,Y 559.156,Z 88.958,A -85,B 0,C 180,E1 -3035.495,E2 -3035.495} C_VEL
LIN {X 0,Y 559.17,Z 88.956,A -85,B 0,C 180,E1 -3038.624,E2 -3038.624} C_VEL
LIN {X 0,Y 559.161,Z 88.963,A -85,B 0,C 180,E1 -3040.926,E2 -3040.926} C_VEL
LIN {X 0,Y 559.163,Z 88.953,A -85,B 0,C 180,E1 -3043.948,E2 -3043.948} C_VEL
LIN {X 0,Y 559.173,Z 88.953,A -85,B 0,C 180,E1 -3046.184,E2 -3046.184} C_VEL
LIN {X 0,Y 559.193,Z 88.952,A -85,B 0,C 180,E1 -3049.134,E2 -3049.134} C_VEL
LIN {X 0,Y 559.203,Z 88.95,A -85,B 0,C 180,E1 -3052.054,E2 -3052.054} C_VEL
LIN {X 0,Y 559.25,Z 88.945,A -85,B 0,C 180,E1 -3054.953,E2 -3054.953} C_VEL
LIN {X 0,Y 559.25,Z 88.944,A -85,B 0,C 180,E1 -3057.84,E2 -3057.84} C_VEL
LIN {X 0,Y 559.269,Z 88.943,A -85,B 0,C 180,E1 -3060.72,E2 -3060.72} C_VEL
LIN {X 0,Y 559.235,Z 88.945,A -85,B 0,C 180,E1 -3062.882,E2 -3062.882} C_VEL
LIN {X 0,Y 559.223,Z 88.95,A -85,B 0,C 180,E1 -3065.77,E2 -3065.77} C_VEL
LIN {X 0,Y 559.186,Z 88.951,A -85,B 0,C 180,E1 -3068.675,E2 -3068.675} C_VEL
LIN {X 0,Y 559.205,Z 88.952,A -85,B 0,C 180,E1 -3071.601,E2 -3071.601} C_VEL
LIN {X 0,Y 559.2,Z 88.949,A -85,B 0,C 180,E1 -3074.596,E2 -3074.596} C_VEL
LIN {X 0,Y 559.14,Z 88.963,A -85,B 0,C 180,E1 -3077.558,E2 -3077.558} C_VEL
LIN {X 0,Y 559.168,Z 88.959,A -85,B 0,C 180,E1 -3079.838,E2 -3079.838} C_VEL
LIN {X 0,Y 559.14,Z 88.958,A -85,B 0,C 180,E1 -3082.153,E2 -3082.153} C_VEL
LIN {X 0,Y 559.175,Z 88.958,A -85,B 0,C 180,E1 -3085.298,E2 -3085.298} C_VEL
LIN {X 0,Y 559.181,Z 88.955,A -85,B 0,C 180,E1 -3087.712,E2 -3087.712} C_VEL
LIN {X 0,Y 559.134,Z 88.957,A -85,B 0,C 180,E1 -3090.603,E2 -3090.603} C_VEL
LIN {X 0,Y 558.473,Z 89.047,A -85,B 0,C 180,E1 -3091.205,E2 -3091.205} C_VEL
LIN {X 0,Y 555.61,Z 89.403,A -85,B 0,C 180,E1 -3092.181,E2 -3092.181} C_VEL
LIN {X 0,Y 553.194,Z 89.702,A -85,B 0,C 180,E1 -3092.967,E2 -3092.967} C_VEL
LIN {X 0,Y 552.167,Z 89.829,A -85,B 0,C 180,E1 -3093.573,E2 -3093.573} C_VEL
LIN {X 0,Y 552.09,Z 89.835,A -85,B 0,C 180,E1 -3093.779,E2 -3093.779} C_VEL
LIN {X 0,Y 552.105,Z 89.836,A -85,B 0,C 180,E1 -3096.747,E2 -3096.747} C_VEL
LIN {X 0,Y 552.128,Z 89.831,A -85,B 0,C 180,E1 -3099.528,E2 -3099.528} C_VEL
LIN {X 0,Y 552.13,Z 89.832,A -85,B 0,C 180,E1 -3102.426,E2 -3102.426} C_VEL
LIN {X 0,Y 552.094,Z 89.834,A -85,B 0,C 180,E1 -3105.563,E2 -3105.563} C_VEL
LIN {X 0,Y 552.121,Z 89.84,A -85,B 0,C 180,E1 -3108.679,E2 -3108.679} C_VEL
LIN {X 0,Y 552.116,Z 89.831,A -85,B 0,C 180,E1 -3111.411,E2 -3111.411} C_VEL
LIN {X 0,Y 552.076,Z 89.84,A -85,B 0,C 180,E1 -3114.156,E2 -3114.156} C_VEL
LIN {X 0,Y 552.117,Z 89.834,A -85,B 0,C 180,E1 -3116.815,E2 -3116.815} C_VEL
LIN {X 0,Y 552.103,Z 89.832,A -85,B 0,C 180,E1 -3119.391,E2 -3119.391} C_VEL
LIN {X 0,Y 552.078,Z 89.839,A -85,B 0,C 180,E1 -3121.9,E2 -3121.9} C_VEL
LIN {X 0,Y 552.124,Z 89.832,A -85,B 0,C 180,E1 -3124.658,E2 -3124.658} C_VEL
LIN {X 0,Y 552.093,Z 89.836,A -85,B 0,C 180,E1 -3127.549,E2 -3127.549} C_VEL
LIN {X 0,Y 552.147,Z 89.833,A -85,B 0,C 180,E1 -3130.375,E2 -3130.375} C_VEL
LIN {X 0,Y 552.134,Z 89.833,A -85,B 0,C 180,E1 -3132.977,E2 -3132.977} C_VEL
LIN {X 0,Y 552.129,Z 89.935,A -85,B 0,C 180,E1 -3133.809,E2 -3133.809} C_VEL
LIN {X 0,Y 553.072,Z 95.989,A -85,B 0,C 180,E1 -3134.828,E2 -3134.828} C_VEL
LIN {X 0,Y 552.725,Z 114.075,A -85,B 0,C 180,E1 -3137.703,E2 -3137.703} C_VEL
LIN {X 0,Y 552.678,Z 120.287,A -85,B 0,C 180,E1 -3138.645,E2 -3138.645} C_VEL
LIN {X 0,Y 554.16,Z 128.33,A -85,B 0,C 180,E1 -3138.8,E2 -3138.8} C_VEL
LIN {X 0,Y 553.743,Z 256.47,A -85,B 0,C 180,E1 -3140.503,E2 -3140.503} C_VEL
LIN {X 0,Y 553.589,Z 270.98,A -85,B 0,C 180,E1 -3140.846,E2 -3140.846} C_VEL
LIN {X 0,Y 553.442,Z 284.792,A -85,B 0,C 180,E1 -3141.327,E2 -3141.327} C_VEL
LIN {X 0,Y 553.182,Z 298.534,A -85,B 0,C 180,E1 -3141.967,E2 -3141.967} C_VEL
LIN {X 0,Y 552.884,Z 310.853,A -85,B 0,C 180,E1 -3142.697,E2 -3142.697} C_VEL
LIN {X 0,Y 552.682,Z 323.256,A -85,B 0,C 180,E1 -3143.612,E2 -3143.612} C_VEL
LIN {X 0,Y 552.414,Z 333.442,A -85,B 0,C 180,E1 -3144.525,E2 -3144.525} C_VEL
LIN {X 0,Y 552.17,Z 343.612,A -85,B 0,C 180,E1 -3145.62,E2 -3145.62} C_VEL
LIN {X 0,Y 552.057,Z 352.023,A -85,B 0,C 180,E1 -3146.716,E2 -3146.716} C_VEL
LIN {X 0,Y 551.896,Z 360.123,A -85,B 0,C 180,E1 -3147.993,E2 -3147.993} C_VEL
LIN {X 0,Y 551.757,Z 366.684,A -85,B 0,C 180,E1 -3149.27,E2 -3149.27} C_VEL
LIN {X 0,Y 551.699,Z 372.527,A -85,B 0,C 180,E1 -3150.73,E2 -3150.73} C_VEL
LIN {X 0,Y 551.657,Z 376.826,A -85,B 0,C 180,E1 -3152.19,E2 -3152.19} C_VEL
LIN {X 0,Y 551.729,Z 379.694,A -85,B 0,C 180,E1 -3153.652,E2 -3153.652} C_VEL
LIN {X 0,Y 551.678,Z 381.207,A -85,B 0,C 180,E1 -3155.116,E2 -3155.116} C_VEL
LIN {X 0,Y 551.747,Z 381.389,A -85,B 0,C 180,E1 -3156.583,E2 -3156.583} C_VEL
LIN {X 0,Y 551.696,Z 380.233,A -85,B 0,C 180,E1 -3158.055,E2 -3158.055} C_VEL
LIN {X 0,Y 551.671,Z 377.704,A -85,B 0,C 180,E1 -3159.533,E2 -3159.533} C_VEL
LIN {X 0,Y 551.761,Z 373.693,A -85,B 0,C 180,E1 -3161.015,E2 -3161.015} C_VEL
LIN {X 0,Y 551.795,Z 368.065,A -85,B 0,C 180,E1 -3162.505,E2 -3162.505} C_VEL
LIN {X 0,Y 551.895,Z 361.669,A -85,B 0,C 180,E1 -3163.814,E2 -3163.814} C_VEL
LIN {X 0,Y 552.009,Z 353.676,A -85,B 0,C 180,E1 -3165.129,E2 -3165.129} C_VEL
LIN {X 0,Y 552.137,Z 345.291,A -85,B 0,C 180,E1 -3166.262,E2 -3166.262} C_VEL
LIN {X 0,Y 552.393,Z 335.06,A -85,B 0,C 180,E1 -3167.404,E2 -3167.404} C_VEL
LIN {X 0,Y 552.642,Z 323.73,A -85,B 0,C 180,E1 -3168.442,E2 -3168.442} C_VEL
LIN {X 0,Y 552.9,Z 311.211,A -85,B 0,C 180,E1 -3169.369,E2 -3169.369} C_VEL
LIN {X 0,Y 553.136,Z 299.691,A -85,B 0,C 180,E1 -3170.063,E2 -3170.063} C_VEL
LIN {X 0,Y 553.377,Z 286.729,A -85,B 0,C 180,E1 -3170.685,E2 -3170.685} C_VEL
LIN {X 0,Y 553.593,Z 272.819,A -85,B 0,C 180,E1 -3171.187,E2 -3171.187} C_VEL
LIN {X 0,Y 553.713,Z 258.385,A -85,B 0,C 180,E1 -3171.549,E2 -3171.549} C_VEL
LIN {X 0,Y 553.871,Z 230.987,A -85,B 0,C 180,E1 -3171.937,E2 -3171.937} C_VEL
LIN {X 0,Y 554.145,Z 127.626,A -85,B 0,C 180,E1 -3173.299,E2 -3173.299} C_VEL
LIN {X 0,Y 552.644,Z 120.035,A -85,B 0,C 180,E1 -3173.451,E2 -3173.451} C_VEL
LIN {X 0,Y 552.925,Z 102.603,A -85,B 0,C 180,E1 -3176.212,E2 -3176.212} C_VEL
LIN {X 0,Y 553.001,Z 94.971,A -85,B 0,C 180,E1 -3177.432,E2 -3177.432} C_VEL
LIN {X 0,Y 552.069,Z 89.846,A -85,B 0,C 180,E1 -3178.32,E2 -3178.32} C_VEL
LIN {X 0,Y 552.072,Z 89.842,A -85,B 0,C 180,E1 -3180.611,E2 -3180.611} C_VEL
LIN {X 0,Y 552.09,Z 89.835,A -85,B 0,C 180,E1 -3183.188,E2 -3183.188} C_VEL
LIN {X 0,Y 552.067,Z 89.846,A -85,B 0,C 180,E1 -3185.845,E2 -3185.845} C_VEL
LIN {X 0,Y 552.088,Z 89.836,A -85,B 0,C 180,E1 -3188.591,E2 -3188.591} C_VEL
LIN {X 0,Y 552.052,Z 89.845,A -85,B 0,C 180,E1 -3191.452,E2 -3191.452} C_VEL
LIN {X 0,Y 552.067,Z 89.837,A -85,B 0,C 180,E1 -3194.528,E2 -3194.528} C_VEL
LIN {X 0,Y 552.084,Z 89.844,A -85,B 0,C 180,E1 -3197.59,E2 -3197.59} C_VEL
LIN {X 0,Y 552.109,Z 89.829,A -85,B 0,C 180,E1 -3200.471,E2 -3200.471} C_VEL
LIN {X 0,Y 552.097,Z 89.842,A -85,B 0,C 180,E1 -3203.318,E2 -3203.318} C_VEL
LIN {X 0,Y 552.1,Z 89.834,A -85,B 0,C 180,E1 -3205.937,E2 -3205.937} C_VEL
LIN {X 0,Y 552.121,Z 89.832,A -85,B 0,C 180,E1 -3208.54,E2 -3208.54} C_VEL
LIN {X 0,Y 552.082,Z 89.839,A -85,B 0,C 180,E1 -3211.446,E2 -3211.446} C_VEL
LIN {X 0,Y 552.081,Z 89.836,A -85,B 0,C 180,E1 -3214.353,E2 -3214.353} C_VEL
LIN {X 0,Y 552.089,Z 89.843,A -85,B 0,C 180,E1 -3216.757,E2 -3216.757} C_VEL
LIN {X 0,Y 552.116,Z 89.835,A -85,B 0,C 180,E1 -3219.119,E2 -3219.119} C_VEL
LIN {X 0,Y 552.088,Z 89.833,A -85,B 0,C 180,E1 -3221.443,E2 -3221.443} C_VEL
LIN {X 0,Y 552.102,Z 89.833,A -85,B 0,C 180,E1 -3223.737,E2 -3223.737} C_VEL
LIN {X 0,Y 552.109,Z 89.834,A -85,B 0,C 180,E1 -3226.004,E2 -3226.004} C_VEL
LIN {X 0,Y 552.16,Z 89.827,A -85,B 0,C 180,E1 -3228.993,E2 -3228.993} C_VEL
LIN {X 0,Y 552.149,Z 89.829,A -85,B 0,C 180,E1 -3231.951,E2 -3231.951} C_VEL
LIN {X 0,Y 552.219,Z 89.818,A -85,B 0,C 180,E1 -3234.889,E2 -3234.889} C_VEL
LIN {X 0,Y 552.223,Z 89.823,A -85,B 0,C 180,E1 -3237.812,E2 -3237.812} C_VEL
LIN {X 0,Y 552.239,Z 89.814,A -85,B 0,C 180,E1 -3240.729,E2 -3240.729} C_VEL
LIN {X 0,Y 552.2,Z 89.82,A -85,B 0,C 180,E1 -3242.918,E2 -3242.918} C_VEL
LIN {X 0,Y 552.188,Z 89.827,A -85,B 0,C 180,E1 -3245.844,E2 -3245.844} C_VEL
LIN {X 0,Y 552.151,Z 89.827,A -85,B 0,C 180,E1 -3248.786,E2 -3248.786} C_VEL
LIN {X 0,Y 552.163,Z 89.83,A -85,B 0,C 180,E1 -3251.75,E2 -3251.75} C_VEL
LIN {X 0,Y 552.129,Z 89.831,A -85,B 0,C 180,E1 -3254.748,E2 -3254.748} C_VEL
LIN {X 0,Y 552.109,Z 89.834,A -85,B 0,C 180,E1 -3257.788,E2 -3257.788} C_VEL
LIN {X 0,Y 552.127,Z 89.828,A -85,B 0,C 180,E1 -3260.101,E2 -3260.101} C_VEL
LIN {X 0,Y 552.091,Z 89.835,A -85,B 0,C 180,E1 -3262.451,E2 -3262.451} C_VEL
LIN {X 0,Y 552.157,Z 89.829,A -85,B 0,C 180,E1 -3265.35,E2 -3265.35} C_VEL
LIN {X 0,Y 552.11,Z 89.832,A -85,B 0,C 180,E1 -3268.098,E2 -3268.098} C_VEL
LIN {X 0,Y 552.108,Z 89.838,A -85,B 0,C 180,E1 -3270.609,E2 -3270.609} C_VEL
LIN {X 0,Y 552.124,Z 89.833,A -85,B 0,C 180,E1 -3273.185,E2 -3273.185} C_VEL
LIN {X 0,Y 552.087,Z 89.834,A -85,B 0,C 180,E1 -3275.844,E2 -3275.844} C_VEL
LIN {X 0,Y 552.122,Z 89.829,A -85,B 0,C 180,E1 -3279.061,E2 -3279.061} C_VEL
LIN {X 0,Y 552.131,Z 89.829,A -85,B 0,C 180,E1 -3281.445,E2 -3281.445} C_VEL
LIN {X 0,Y 552.094,Z 89.839,A -85,B 0,C 180,E1 -3284.532,E2 -3284.532} C_VEL
LIN {X 0,Y 552.13,Z 89.831,A -85,B 0,C 180,E1 -3287.585,E2 -3287.585} C_VEL
LIN {X 0,Y 552.133,Z 89.832,A -85,B 0,C 180,E1 -3290.473,E2 -3290.473} C_VEL
LIN {X 0,Y 552.108,Z 89.833,A -85,B 0,C 180,E1 -3293.317,E2 -3293.317} C_VEL
LIN {X 0,Y 552.128,Z 89.837,A -85,B 0,C 180,E1 -3295.939,E2 -3295.939} C_VEL
LIN {X 0,Y 552.121,Z 89.831,A -85,B 0,C 180,E1 -3298.541,E2 -3298.541} C_VEL
LIN {X 0,Y 552.126,Z 89.837,A -85,B 0,C 180,E1 -3301.438,E2 -3301.438} C_VEL
LIN {X 0,Y 552.132,Z 89.834,A -85,B 0,C 180,E1 -3304.356,E2 -3304.356} C_VEL
LIN {X 0,Y 552.196,Z 89.852,A -85,B 0,C 180,E1 -3305.127,E2 -3305.127} C_VEL
LIN {X 0,Y 553.486,Z 97.207,A -85,B 0,C 180,E1 -3306.229,E2 -3306.229} C_VEL
LIN {X 0,Y 553.139,Z 116.861,A -85,B 0,C 180,E1 -3308.965,E2 -3308.965} C_VEL
LIN {X 0,Y 552.808,Z 137.944,A -85,B 0,C 180,E1 -3311.852,E2 -3311.852} C_VEL
LIN {X 0,Y 552.728,Z 143.3,A -85,B 0,C 180,E1 -3312.579,E2 -3312.579} C_VEL
LIN {X 0,Y 554.195,Z 152.274,A -85,B 0,C 180,E1 -3312.752,E2 -3312.752} C_VEL
LIN {X 0,Y 553.714,Z 281.619,A -85,B 0,C 180,E1 -3314.471,E2 -3314.471} C_VEL
LIN {X 0,Y 553.561,Z 296.182,A -85,B 0,C 180,E1 -3314.821,E2 -3314.821} C_VEL
LIN {X 0,Y 553.345,Z 310.626,A -85,B 0,C 180,E1 -3315.331,E2 -3315.331} C_VEL
LIN {X 0,Y 553.147,Z 323.462,A -85,B 0,C 180,E1 -3315.937,E2 -3315.937} C_VEL
LIN {X 0,Y 552.869,Z 335.959,A -85,B 0,C 180,E1 -3316.679,E2 -3316.679} C_VEL
LIN {X 0,Y 552.624,Z 348.557,A -85,B 0,C 180,E1 -3317.607,E2 -3317.607} C_VEL
LIN {X 0,Y 552.383,Z 359.299,A -85,B 0,C 180,E1 -3318.577,E2 -3318.577} C_VEL
LIN {X 0,Y 552.179,Z 369.845,A -85,B 0,C 180,E1 -3319.736,E2 -3319.736} C_VEL
LIN {X 0,Y 552.032,Z 378.173,A -85,B 0,C 180,E1 -3320.843,E2 -3320.843} C_VEL
LIN {X 0,Y 551.913,Z 386.126,A -85,B 0,C 180,E1 -3322.132,E2 -3322.132} C_VEL
LIN {X 0,Y 551.822,Z 392.527,A -85,B 0,C 180,E1 -3323.418,E2 -3323.418} C_VEL
LIN {X 0,Y 551.791,Z 396.96,A -85,B 0,C 180,E1 -3324.518,E2 -3324.518} C_VEL
LIN {X 0,Y 551.76,Z 400.443,A -85,B 0,C 180,E1 -3325.617,E2 -3325.617} C_VEL
LIN {X 0,Y 551.719,Z 403.832,A -85,B 0,C 180,E1 -3327.079,E2 -3327.079} C_VEL
LIN {X 0,Y 551.641,Z 405.835,A -85,B 0,C 180,E1 -3328.54,E2 -3328.54} C_VEL
LIN {X 0,Y 551.639,Z 406.5,A -85,B 0,C 180,E1 -3330,E2 -3330} C_VEL
LIN {X 0,Y 551.641,Z 405.836,A -85,B 0,C 180,E1 -3331.46,E2 -3331.46} C_VEL
LIN {X 0,Y 551.719,Z 403.836,A -85,B 0,C 180,E1 -3332.921,E2 -3332.921} C_VEL
LIN {X 0,Y 551.76,Z 400.447,A -85,B 0,C 180,E1 -3334.383,E2 -3334.383} C_VEL
LIN {X 0,Y 551.823,Z 395.568,A -85,B 0,C 180,E1 -3335.848,E2 -3335.848} C_VEL
LIN {X 0,Y 551.832,Z 389.054,A -85,B 0,C 180,E1 -3337.317,E2 -3337.317} C_VEL
LIN {X 0,Y 551.962,Z 381.804,A -85,B 0,C 180,E1 -3338.604,E2 -3338.604} C_VEL
LIN {X 0,Y 552.116,Z 372.822,A -85,B 0,C 180,E1 -3339.895,E2 -3339.895} C_VEL
LIN {X 0,Y 552.346,Z 363.361,A -85,B 0,C 180,E1 -3341.003,E2 -3341.003} C_VEL
LIN {X 0,Y 552.503,Z 352.877,A -85,B 0,C 180,E1 -3342.022,E2 -3342.022} C_VEL
LIN {X 0,Y 552.715,Z 341.312,A -85,B 0,C 180,E1 -3342.95,E2 -3342.95} C_VEL
LIN {X 0,Y 553.021,Z 328.486,A -85,B 0,C 180,E1 -3343.785,E2 -3343.785} C_VEL
LIN {X 0,Y 553.241,Z 315.959,A -85,B 0,C 180,E1 -3344.436,E2 -3344.436} C_VEL
LIN {X 0,Y 553.489,Z 302.813,A -85,B 0,C 180,E1 -3344.965,E2 -3344.965} C_VEL
LIN {X 0,Y 553.652,Z 288.67,A -85,B 0,C 180,E1 -3345.38,E2 -3345.38} C_VEL
LIN {X 0,Y 553.77,Z 274.345,A -85,B 0,C 180,E1 -3345.646,E2 -3345.646} C_VEL
LIN {X 0,Y 554.139,Z 151.442,A -85,B 0,C 180,E1 -3347.261,E2 -3347.261} C_VEL
LIN {X 0,Y 552.71,Z 143.345,A -85,B 0,C 180,E1 -3347.417,E2 -3347.417} C_VEL
LIN {X 0,Y 553.079,Z 122.506,A -85,B 0,C 180,E1 -3350.259,E2 -3350.259} C_VEL
LIN {X 0,Y 553.536,Z 98.838,A -85,B 0,C 180,E1 -3353.541,E2 -3353.541} C_VEL
LIN {X 0,Y 553.092,Z 94.38,A -85,B 0,C 180,E1 -3354.192,E2 -3354.192} C_VEL
LIN {X 0,Y 552.183,Z 89.83,A -85,B 0,C 180,E1 -3354.912,E2 -3354.912} C_VEL
LIN {X 0,Y 552.121,Z 89.837,A -85,B 0,C 180,E1 -3358.098,E2 -3358.098} C_VEL
LIN {X 0,Y 552.103,Z 89.838,A -85,B 0,C 180,E1 -3360.609,E2 -3360.609} C_VEL
LIN {X 0,Y 552.116,Z 89.831,A -85,B 0,C 180,E1 -3363.186,E2 -3363.186} C_VEL
LIN {X 0,Y 552.086,Z 89.84,A -85,B 0,C 180,E1 -3365.843,E2 -3365.843} C_VEL
LIN {X 0,Y 552.125,Z 89.83,A -85,B 0,C 180,E1 -3369.062,E2 -3369.062} C_VEL
LIN {X 0,Y 552.136,Z 89.831,A -85,B 0,C 180,E1 -3371.444,E2 -3371.444} C_VEL
LIN {X 0,Y 552.095,Z 89.834,A -85,B 0,C 180,E1 -3374.532,E2 -3374.532} C_VEL
LIN {X 0,Y 552.131,Z 89.836,A -85,B 0,C 180,E1 -3377.584,E2 -3377.584} C_VEL
LIN {X 0,Y 552.129,Z 89.829,A -85,B 0,C 180,E1 -3380.473,E2 -3380.473} C_VEL
LIN {X 0,Y 552.105,Z 89.838,A -85,B 0,C 180,E1 -3383.317,E2 -3383.317} C_VEL
LIN {X 0,Y 552.127,Z 89.832,A -85,B 0,C 180,E1 -3385.939,E2 -3385.939} C_VEL
LIN {X 0,Y 552.118,Z 89.831,A -85,B 0,C 180,E1 -3388.541,E2 -3388.541} C_VEL
LIN {X 0,Y 552.124,Z 89.836,A -85,B 0,C 180,E1 -3391.438,E2 -3391.438} C_VEL
LIN {X 0,Y 552.13,Z 89.829,A -85,B 0,C 180,E1 -3394.356,E2 -3394.356} C_VEL
LIN {X 0,Y 552.098,Z 89.838,A -85,B 0,C 180,E1 -3396.758,E2 -3396.758} C_VEL
LIN {X 0,Y 552.118,Z 89.838,A -85,B 0,C 180,E1 -3399.12,E2 -3399.12} C_VEL
LIN {X 0,Y 552.12,Z 89.833,A -85,B 0,C 180,E1 -3401.444,E2 -3401.444} C_VEL
LIN {X 0,Y 552.113,Z 89.831,A -85,B 0,C 180,E1 -3403.737,E2 -3403.737} C_VEL
LIN {X 0,Y 552.136,Z 89.829,A -85,B 0,C 180,E1 -3406.005,E2 -3406.005} C_VEL
LIN {X 0,Y 552.161,Z 89.83,A -85,B 0,C 180,E1 -3408.993,E2 -3408.993} C_VEL
LIN {X 0,Y 552.157,Z 89.827,A -85,B 0,C 180,E1 -3411.952,E2 -3411.952} C_VEL
LIN {X 0,Y 552.225,Z 89.821,A -85,B 0,C 180,E1 -3414.889,E2 -3414.889} C_VEL
LIN {X 0,Y 552.222,Z 89.819,A -85,B 0,C 180,E1 -3417.812,E2 -3417.812} C_VEL
LIN {X 0,Y 552.24,Z 89.818,A -85,B 0,C 180,E1 -3420.729,E2 -3420.729} C_VEL
LIN {X 0,Y 552.202,Z 89.821,A -85,B 0,C 180,E1 -3422.918,E2 -3422.918} C_VEL
LIN {X 0,Y 552.191,Z 89.827,A -85,B 0,C 180,E1 -3425.844,E2 -3425.844} C_VEL
LIN {X 0,Y 552.157,Z 89.826,A -85,B 0,C 180,E1 -3428.786,E2 -3428.786} C_VEL
LIN {X 0,Y 552.163,Z 89.832,A -85,B 0,C 180,E1 -3431.751,E2 -3431.751} C_VEL
LIN {X 0,Y 552.136,Z 89.828,A -85,B 0,C 180,E1 -3434.749,E2 -3434.749} C_VEL
LIN {X 0,Y 552.097,Z 89.842,A -85,B 0,C 180,E1 -3437.789,E2 -3437.789} C_VEL
LIN {X 0,Y 552.128,Z 89.832,A -85,B 0,C 180,E1 -3440.101,E2 -3440.101} C_VEL
LIN {X 0,Y 552.091,Z 89.834,A -85,B 0,C 180,E1 -3442.451,E2 -3442.451} C_VEL
LIN {X 0,Y 552.155,Z 89.834,A -85,B 0,C 180,E1 -3445.351,E2 -3445.351} C_VEL
LIN {X 0,Y 552.106,Z 89.833,A -85,B 0,C 180,E1 -3448.099,E2 -3448.099} C_VEL
LIN {X 0,Y 552.098,Z 89.834,A -85,B 0,C 180,E1 -3450.61,E2 -3450.61} C_VEL
LIN {X 0,Y 552.107,Z 89.841,A -85,B 0,C 180,E1 -3453.187,E2 -3453.187} C_VEL
LIN {X 0,Y 552.09,Z 89.835,A -85,B 0,C 180,E1 -3453.779,E2 -3453.779} C_VEL
LIN {X 0,Y 551.45,Z 89.915,A -85,B 0,C 180,E1 -3454.387,E2 -3454.387} C_VEL
LIN {X 0,Y 548.637,Z 90.27,A -85,B 0,C 180,E1 -3455.376,E2 -3455.376} C_VEL
LIN {X 0,Y 546.228,Z 90.573,A -85,B 0,C 180,E1 -3456.171,E2 -3456.171} C_VEL
LIN {X 0,Y 545.164,Z 90.704,A -85,B 0,C 180,E1 -3456.785,E2 -3456.785} C_VEL
LIN {X 0,Y 545.062,Z 90.716,A -85,B 0,C 180,E1 -3456.993,E2 -3456.993} C_VEL
LIN {X 0,Y 545.065,Z 90.709,A -85,B 0,C 180,E1 -3460.143,E2 -3460.143} C_VEL
LIN {X 0,Y 545.079,Z 90.713,A -85,B 0,C 180,E1 -3463.107,E2 -3463.107} C_VEL
LIN {X 0,Y 545.05,Z 90.713,A -85,B 0,C 180,E1 -3466.227,E2 -3466.227} C_VEL
LIN {X 0,Y 545.081,Z 90.713,A -85,B 0,C 180,E1 -3468.886,E2 -3468.886} C_VEL
LIN {X 0,Y 545.079,Z 90.714,A -85,B 0,C 180,E1 -3470.818,E2 -3470.818} C_VEL
LIN {X 0,Y 545.035,Z 90.713,A -85,B 0,C 180,E1 -3473.619,E2 -3473.619} C_VEL
LIN {X 0,Y 545.067,Z 90.716,A -85,B 0,C 180,E1 -3476.328,E2 -3476.328} C_VEL
LIN {X 0,Y 545.068,Z 90.71,A -85,B 0,C 180,E1 -3478.952,E2 -3478.952} C_VEL
LIN {X 0,Y 545.077,Z 90.708,A -85,B 0,C 180,E1 -3481.506,E2 -3481.506} C_VEL
LIN {X 0,Y 545.095,Z 90.707,A -85,B 0,C 180,E1 -3484.82,E2 -3484.82} C_VEL
LIN {X 0,Y 545.037,Z 90.713,A -85,B 0,C 180,E1 -3487.242,E2 -3487.242} C_VEL
LIN {X 0,Y 545.119,Z 90.708,A -85,B 0,C 180,E1 -3490.415,E2 -3490.415} C_VEL
LIN {X 0,Y 545.08,Z 90.743,A -85,B 0,C 180,E1 -3493.618,E2 -3493.618} C_VEL
LIN {X 0,Y 546.105,Z 96.797,A -85,B 0,C 180,E1 -3494.656,E2 -3494.656} C_VEL
LIN {X 0,Y 545.784,Z 114.749,A -85,B 0,C 180,E1 -3497.544,E2 -3497.544} C_VEL
LIN {X 0,Y 545.705,Z 120.182,A -85,B 0,C 180,E1 -3498.41,E2 -3498.41} C_VEL
LIN {X 0,Y 547.418,Z 129.696,A -85,B 0,C 180,E1 -3498.597,E2 -3498.597} C_VEL
LIN {X 0,Y 546.915,Z 257.083,A -85,B 0,C 180,E1 -3500.314,E2 -3500.314} C_VEL
LIN {X 0,Y 546.755,Z 271.424,A -85,B 0,C 180,E1 -3500.661,E2 -3500.661} C_VEL
LIN {X 0,Y 546.569,Z 285.722,A -85,B 0,C 180,E1 -3501.171,E2 -3501.171} C_VEL
LIN {X 0,Y 546.292,Z 298.433,A -85,B 0,C 180,E1 -3501.772,E2 -3501.772} C_VEL
LIN {X 0,Y 545.954,Z 310.944,A -85,B 0,C 180,E1 -3502.52,E2 -3502.52} C_VEL
LIN {X 0,Y 545.724,Z 323.246,A -85,B 0,C 180,E1 -3503.437,E2 -3503.437} C_VEL
LIN {X 0,Y 545.412,Z 334.414,A -85,B 0,C 180,E1 -3504.454,E2 -3504.454} C_VEL
LIN {X 0,Y 545.142,Z 344.413,A -85,B 0,C 180,E1 -3505.564,E2 -3505.564} C_VEL
LIN {X 0,Y 545.009,Z 352.727,A -85,B 0,C 180,E1 -3506.673,E2 -3506.673} C_VEL
LIN {X 0,Y 544.83,Z 360.694,A -85,B 0,C 180,E1 -3507.967,E2 -3507.967} C_VEL
LIN {X 0,Y 544.674,Z 367.139,A -85,B 0,C 180,E1 -3509.261,E2 -3509.261} C_VEL
LIN {X 0,Y 544.607,Z 372.872,A -85,B 0,C 180,E1 -3510.74,E2 -3510.74} C_VEL
LIN {X 0,Y 544.572,Z 377.073,A -85,B 0,C 180,E1 -3512.219,E2 -3512.219} C_VEL
LIN {X 0,Y 544.643,Z 379.851,A -85,B 0,C 180,E1 -3513.699,E2 -3513.699} C_VEL
LIN {X 0,Y 544.598,Z 381.289,A -85,B 0,C 180,E1 -3515.183,E2 -3515.183} C_VEL
LIN {X 0,Y 544.651,Z 381.4,A -85,B 0,C 180,E1 -3516.669,E2 -3516.669} C_VEL
LIN {X 0,Y 544.612,Z 380.182,A -85,B 0,C 180,E1 -3518.161,E2 -3518.161} C_VEL
LIN {X 0,Y 544.598,Z 377.578,A -85,B 0,C 180,E1 -3519.658,E2 -3519.658} C_VEL
LIN {X 0,Y 544.675,Z 373.503,A -85,B 0,C 180,E1 -3521.16,E2 -3521.16} C_VEL
LIN {X 0,Y 544.716,Z 367.824,A -85,B 0,C 180,E1 -3522.67,E2 -3522.67} C_VEL
LIN {X 0,Y 544.82,Z 361.373,A -85,B 0,C 180,E1 -3523.997,E2 -3523.997} C_VEL
LIN {X 0,Y 544.974,Z 353.305,A -85,B 0,C 180,E1 -3525.33,E2 -3525.33} C_VEL
LIN {X 0,Y 545.158,Z 344.809,A -85,B 0,C 180,E1 -3526.476,E2 -3526.476} C_VEL
LIN {X 0,Y 545.392,Z 335.468,A -85,B 0,C 180,E1 -3527.526,E2 -3527.526} C_VEL
LIN {X 0,Y 545.692,Z 324.065,A -85,B 0,C 180,E1 -3528.588,E2 -3528.588} C_VEL
LIN {X 0,Y 545.947,Z 312.65,A -85,B 0,C 180,E1 -3529.456,E2 -3529.456} C_VEL
LIN {X 0,Y 546.254,Z 299.593,A -85,B 0,C 180,E1 -3530.257,E2 -3530.257} C_VEL
LIN {X 0,Y 546.504,Z 287.232,A -85,B 0,C 180,E1 -3530.858,E2 -3530.858} C_VEL
LIN {X 0,Y 546.744,Z 273.443,A -85,B 0,C 180,E1 -3531.367,E2 -3531.367} C_VEL
LIN {X 0,Y 546.884,Z 259.244,A -85,B 0,C 180,E1 -3531.732,E2 -3531.732} C_VEL
LIN {X 0,Y 547.013,Z 236.241,A -85,B 0,C 180,E1 -3532.073,E2 -3532.073} C_VEL
LIN {X 0,Y 547.415,Z 128.904,A -85,B 0,C 180,E1 -3533.503,E2 -3533.503} C_VEL
LIN {X 0,Y 545.7,Z 120.066,A -85,B 0,C 180,E1 -3533.702,E2 -3533.702} C_VEL
LIN {X 0,Y 546.015,Z 103.441,A -85,B 0,C 180,E1 -3536.364,E2 -3536.364} C_VEL
LIN {X 0,Y 545.989,Z 95.803,A -85,B 0,C 180,E1 -3537.606,E2 -3537.606} C_VEL
LIN {X 0,Y 545.043,Z 90.721,A -85,B 0,C 180,E1 -3538.496,E2 -3538.496} C_VEL
LIN {X 0,Y 545.044,Z 90.718,A -85,B 0,C 180,E1 -3541.676,E2 -3541.676} C_VEL
LIN {X 0,Y 545.041,Z 90.715,A -85,B 0,C 180,E1 -3544.566,E2 -3544.566} C_VEL
LIN {X 0,Y 545.009,Z 90.718,A -85,B 0,C 180,E1 -3547.306,E2 -3547.306} C_VEL
LIN {X 0,Y 545.009,Z 90.721,A -85,B 0,C 180,E1 -3550.148,E2 -3550.148} C_VEL
LIN {X 0,Y 545.01,Z 90.717,A -85,B 0,C 180,E1 -3552.69,E2 -3552.69} C_VEL
LIN {X 0,Y 545.018,Z 90.719,A -85,B 0,C 180,E1 -3555.172,E2 -3555.172} C_VEL
LIN {X 0,Y 545.034,Z 90.717,A -85,B 0,C 180,E1 -3557.892,E2 -3557.892} C_VEL
LIN {X 0,Y 545.07,Z 90.707,A -85,B 0,C 180,E1 -3560.817,E2 -3560.817} C_VEL
LIN {X 0,Y 545.032,Z 90.717,A -85,B 0,C 180,E1 -3563.619,E2 -3563.619} C_VEL
LIN {X 0,Y 545.048,Z 90.712,A -85,B 0,C 180,E1 -3566.327,E2 -3566.327} C_VEL
LIN {X 0,Y 545.062,Z 90.717,A -85,B 0,C 180,E1 -3568.952,E2 -3568.952} C_VEL
LIN {X 0,Y 545.042,Z 90.715,A -85,B 0,C 180,E1 -3571.504,E2 -3571.504} C_VEL
LIN {X 0,Y 545.043,Z 90.711,A -85,B 0,C 180,E1 -3573.997,E2 -3573.997} C_VEL
LIN {X 0,Y 545.071,Z 90.713,A -85,B 0,C 180,E1 -3576.44,E2 -3576.44} C_VEL
LIN {X 0,Y 545.091,Z 90.707,A -85,B 0,C 180,E1 -3579.628,E2 -3579.628} C_VEL
LIN {X 0,Y 545.064,Z 90.716,A -85,B 0,C 180,E1 -3582.749,E2 -3582.749} C_VEL
LIN {X 0,Y 545.067,Z 90.71,A -85,B 0,C 180,E1 -3585.819,E2 -3585.819} C_VEL
LIN {X 0,Y 545.117,Z 90.706,A -85,B 0,C 180,E1 -3588.849,E2 -3588.849} C_VEL
LIN {X 0,Y 545.097,Z 90.706,A -85,B 0,C 180,E1 -3591.846,E2 -3591.846} C_VEL
LIN {X 0,Y 545.196,Z 90.693,A -85,B 0,C 180,E1 -3594.823,E2 -3594.823} C_VEL
LIN {X 0,Y 545.195,Z 90.698,A -85,B 0,C 180,E1 -3597.784,E2 -3597.784} C_VEL
LIN {X 0,Y 545.209,Z 90.69,A -85,B 0,C 180,E1 -3600.738,E2 -3600.738} C_VEL
LIN {X 0,Y 545.167,Z 90.697,A -85,B 0,C 180,E1 -3602.956,E2 -3602.956} C_VEL
LIN {X 0,Y 545.138,Z 90.704,A -85,B 0,C 180,E1 -3605.92,E2 -3605.92} C_VEL
LIN {X 0,Y 545.109,Z 90.705,A -85,B 0,C 180,E1 -3608.9,E2 -3608.9} C_VEL
LIN {X 0,Y 545.107,Z 90.707,A -85,B 0,C 180,E1 -3611.905,E2 -3611.905} C_VEL
LIN {X 0,Y 545.082,Z 90.71,A -85,B 0,C 180,E1 -3614.944,E2 -3614.944} C_VEL
LIN {X 0,Y 545.077,Z 90.708,A -85,B 0,C 180,E1 -3618.026,E2 -3618.026} C_VEL
LIN {X 0,Y 545.093,Z 90.705,A -85,B 0,C 180,E1 -3620.372,E2 -3620.372} C_VEL
LIN {X 0,Y 545.08,Z 90.709,A -85,B 0,C 180,E1 -3623.559,E2 -3623.559} C_VEL
LIN {X 0,Y 545.081,Z 90.707,A -85,B 0,C 180,E1 -3626,E2 -3626} C_VEL
LIN {X 0,Y 545.09,Z 90.713,A -85,B 0,C 180,E1 -3628.748,E2 -3628.748} C_VEL
LIN {X 0,Y 545.06,Z 90.71,A -85,B 0,C 180,E1 -3631.679,E2 -3631.679} C_VEL
LIN {X 0,Y 545.075,Z 90.716,A -85,B 0,C 180,E1 -3634.564,E2 -3634.564} C_VEL
LIN {X 0,Y 545.036,Z 90.714,A -85,B 0,C 180,E1 -3637.304,E2 -3637.304} C_VEL
LIN {X 0,Y 545.066,Z 90.71,A -85,B 0,C 180,E1 -3640.143,E2 -3640.143} C_VEL
LIN {X 0,Y 545.079,Z 90.708,A -85,B 0,C 180,E1 -3643.107,E2 -3643.107} C_VEL
LIN {X 0,Y 545.067,Z 90.717,A -85,B 0,C 180,E1 -3646.224,E2 -3646.224} C_VEL
LIN {X 0,Y 545.092,Z 90.707,A -85,B 0,C 180,E1 -3648.886,E2 -3648.886} C_VEL
LIN {X 0,Y 545.056,Z 90.715,A -85,B 0,C 180,E1 -3651.763,E2 -3651.763} C_VEL
LIN {X 0,Y 545.038,Z 90.714,A -85,B 0,C 180,E1 -3654.532,E2 -3654.532} C_VEL
LIN {X 0,Y 545.07,Z 90.708,A -85,B 0,C 180,E1 -3657.212,E2 -3657.212} C_VEL
LIN {X 0,Y 545.065,Z 90.717,A -85,B 0,C 180,E1 -3659.811,E2 -3659.811} C_VEL
LIN {X 0,Y 545.091,Z 90.71,A -85,B 0,C 180,E1 -3662.344,E2 -3662.344} C_VEL
LIN {X 0,Y 545.155,Z 90.855,A -85,B 0,C 180,E1 -3664.95,E2 -3664.95} C_VEL
LIN {X 0,Y 546.468,Z 97.307,A -85,B 0,C 180,E1 -3665.94,E2 -3665.94} C_VEL
LIN {X 0,Y 546.439,Z 108.153,A -85,B 0,C 180,E1 -3667.487,E2 -3667.487} C_VEL
LIN {X 0,Y 545.971,Z 129.345,A -85,B 0,C 180,E1 -3670.447,E2 -3670.447} C_VEL
LIN {X 0,Y 545.745,Z 143.185,A -85,B 0,C 180,E1 -3672.356,E2 -3672.356} C_VEL
LIN {X 0,Y 547.443,Z 153.917,A -85,B 0,C 180,E1 -3672.557,E2 -3672.557} C_VEL
LIN {X 0,Y 546.881,Z 281.44,A -85,B 0,C 180,E1 -3674.272,E2 -3674.272} C_VEL
LIN {X 0,Y 546.72,Z 295.848,A -85,B 0,C 180,E1 -3674.621,E2 -3674.621} C_VEL
LIN {X 0,Y 546.506,Z 309.322,A -85,B 0,C 180,E1 -3675.096,E2 -3675.096} C_VEL
LIN {X 0,Y 546.245,Z 321.52,A -85,B 0,C 180,E1 -3675.66,E2 -3675.66} C_VEL
LIN {X 0,Y 545.938,Z 334.358,A -85,B 0,C 180,E1 -3676.412,E2 -3676.412} C_VEL
LIN {X 0,Y 545.66,Z 346.032,A -85,B 0,C 180,E1 -3677.258,E2 -3677.258} C_VEL
LIN {X 0,Y 545.464,Z 356.783,A -85,B 0,C 180,E1 -3678.202,E2 -3678.202} C_VEL
LIN {X 0,Y 545.231,Z 366.517,A -85,B 0,C 180,E1 -3679.228,E2 -3679.228} C_VEL
LIN {X 0,Y 545.015,Z 375.407,A -85,B 0,C 180,E1 -3680.35,E2 -3680.35} C_VEL
LIN {X 0,Y 544.873,Z 383.928,A -85,B 0,C 180,E1 -3681.656,E2 -3681.656} C_VEL
LIN {X 0,Y 544.736,Z 390.794,A -85,B 0,C 180,E1 -3682.96,E2 -3682.96} C_VEL
LIN {X 0,Y 544.731,Z 395.528,A -85,B 0,C 180,E1 -3684.076,E2 -3684.076} C_VEL
LIN {X 0,Y 544.654,Z 400.431,A -85,B 0,C 180,E1 -3685.56,E2 -3685.56} C_VEL
LIN {X 0,Y 544.646,Z 403.831,A -85,B 0,C 180,E1 -3687.041,E2 -3687.041} C_VEL
LIN {X 0,Y 544.542,Z 405.835,A -85,B 0,C 180,E1 -3688.521,E2 -3688.521} C_VEL
LIN {X 0,Y 544.539,Z 406.5,A -85,B 0,C 180,E1 -3690,E2 -3690} C_VEL
LIN {X 0,Y 544.542,Z 405.837,A -85,B 0,C 180,E1 -3691.479,E2 -3691.479} C_VEL
LIN {X 0,Y 544.646,Z 403.836,A -85,B 0,C 180,E1 -3692.959,E2 -3692.959} C_VEL
LIN {X 0,Y 544.654,Z 400.435,A -85,B 0,C 180,E1 -3694.44,E2 -3694.44} C_VEL
LIN {X 0,Y 544.736,Z 395.528,A -85,B 0,C 180,E1 -3695.924,E2 -3695.924} C_VEL
LIN {X 0,Y 544.736,Z 390.795,A -85,B 0,C 180,E1 -3697.04,E2 -3697.04} C_VEL
LIN {X 0,Y 544.872,Z 383.932,A -85,B 0,C 180,E1 -3698.343,E2 -3698.343} C_VEL
LIN {X 0,Y 545.014,Z 375.412,A -85,B 0,C 180,E1 -3699.65,E2 -3699.65} C_VEL
LIN {X 0,Y 545.232,Z 366.524,A -85,B 0,C 180,E1 -3700.772,E2 -3700.772} C_VEL
LIN {X 0,Y 545.454,Z 355.757,A -85,B 0,C 180,E1 -3701.897,E2 -3701.897} C_VEL
LIN {X 0,Y 545.74,Z 343.688,A -85,B 0,C 180,E1 -3702.929,E2 -3702.929} C_VEL
LIN {X 0,Y 546.018,Z 331.487,A -85,B 0,C 180,E1 -3703.775,E2 -3703.775} C_VEL
LIN {X 0,Y 546.274,Z 319.753,A -85,B 0,C 180,E1 -3704.434,E2 -3704.434} C_VEL
LIN {X 0,Y 546.603,Z 306.293,A -85,B 0,C 180,E1 -3705.025,E2 -3705.025} C_VEL
LIN {X 0,Y 546.733,Z 292.816,A -85,B 0,C 180,E1 -3705.467,E2 -3705.467} C_VEL
LIN {X 0,Y 546.919,Z 278.696,A -85,B 0,C 180,E1 -3705.775,E2 -3705.775} C_VEL
LIN {X 0,Y 547.43,Z 152.824,A -85,B 0,C 180,E1 -3707.458,E2 -3707.458} C_VEL
LIN {X 0,Y 545.747,Z 143.075,A -85,B 0,C 180,E1 -3707.661,E2 -3707.661} C_VEL
LIN {X 0,Y 546.139,Z 122.343,A -85,B 0,C 180,E1 -3710.528,E2 -3710.528} C_VEL
LIN {X 0,Y 546.646,Z 99.298,A -85,B 0,C 180,E1 -3713.772,E2 -3713.772} C_VEL
LIN {X 0,Y 545.59,Z 92.834,A -85,B 0,C 180,E1 -3714.749,E2 -3714.749} C_VEL
LIN {X 0,Y 545.122,Z 90.708,A -85,B 0,C 180,E1 -3715.103,E2 -3715.103} C_VEL
LIN {X 0,Y 545.09,Z 90.709,A -85,B 0,C 180,E1 -3717.656,E2 -3717.656} C_VEL
LIN {X 0,Y 545.078,Z 90.717,A -85,B 0,C 180,E1 -3720.246,E2 -3720.246} C_VEL
LIN {X 0,Y 545.08,Z 90.707,A -85,B 0,C 180,E1 -3723.062,E2 -3723.062} C_VEL
LIN {X 0,Y 545.034,Z 90.716,A -85,B 0,C 180,E1 -3725.673,E2 -3725.673} C_VEL
LIN {X 0,Y 545.055,Z 90.716,A -85,B 0,C 180,E1 -3728.237,E2 -3728.237} C_VEL
LIN {X 0,Y 545.094,Z 90.706,A -85,B 0,C 180,E1 -3731.113,E2 -3731.113} C_VEL
LIN {X 0,Y 545.058,Z 90.715,A -85,B 0,C 180,E1 -3734.129,E2 -3734.129} C_VEL
LIN {X 0,Y 545.087,Z 90.707,A -85,B 0,C 180,E1 -3736.894,E2 -3736.894} C_VEL
LIN {X 0,Y 545.065,Z 90.715,A -85,B 0,C 180,E1 -3739.857,E2 -3739.857} C_VEL
LIN {X 0,Y 545.069,Z 90.711,A -85,B 0,C 180,E1 -3743.074,E2 -3743.074} C_VEL
LIN {X 0,Y 545.068,Z 90.709,A -85,B 0,C 180,E1 -3746.328,E2 -3746.328} C_VEL
LIN {X 0,Y 545.066,Z 90.713,A -85,B 0,C 180,E1 -3748.952,E2 -3748.952} C_VEL
LIN {X 0,Y 545.1,Z 90.71,A -85,B 0,C 180,E1 -3751.508,E2 -3751.508} C_VEL
LIN {X 0,Y 545.095,Z 90.707,A -85,B 0,C 180,E1 -3754.491,E2 -3754.491} C_VEL
LIN {X 0,Y 545.037,Z 90.719,A -85,B 0,C 180,E1 -3757.242,E2 -3757.242} C_VEL
LIN {X 0,Y 545.115,Z 90.705,A -85,B 0,C 180,E1 -3760.415,E2 -3760.415} C_VEL
LIN {X 0,Y 545.07,Z 90.71,A -85,B 0,C 180,E1 -3763.521,E2 -3763.521} C_VEL
LIN {X 0,Y 545.095,Z 90.705,A -85,B 0,C 180,E1 -3765.82,E2 -3765.82} C_VEL
LIN {X 0,Y 545.117,Z 90.709,A -85,B 0,C 180,E1 -3768.849,E2 -3768.849} C_VEL
LIN {X 0,Y 545.127,Z 90.702,A -85,B 0,C 180,E1 -3771.847,E2 -3771.847} C_VEL
LIN {X 0,Y 545.201,Z 90.696,A -85,B 0,C 180,E1 -3774.823,E2 -3774.823} C_VEL
LIN {X 0,Y 545.194,Z 90.695,A -85,B 0,C 180,E1 -3777.784,E2 -3777.784} C_VEL
LIN {X 0,Y 545.21,Z 90.694,A -85,B 0,C 180,E1 -3780.739,E2 -3780.739} C_VEL
LIN {X 0,Y 545.169,Z 90.697,A -85,B 0,C 180,E1 -3782.956,E2 -3782.956} C_VEL
LIN {X 0,Y 545.161,Z 90.703,A -85,B 0,C 180,E1 -3785.92,E2 -3785.92} C_VEL
LIN {X 0,Y 545.116,Z 90.703,A -85,B 0,C 180,E1 -3788.9,E2 -3788.9} C_VEL
LIN {X 0,Y 545.135,Z 90.71,A -85,B 0,C 180,E1 -3791.904,E2 -3791.904} C_VEL
LIN {X 0,Y 545.085,Z 90.707,A -85,B 0,C 180,E1 -3794.944,E2 -3794.944} C_VEL
LIN {X 0,Y 545.062,Z 90.714,A -85,B 0,C 180,E1 -3798.027,E2 -3798.027} C_VEL
LIN {X 0,Y 545.093,Z 90.706,A -85,B 0,C 180,E1 -3800.372,E2 -3800.372} C_VEL
LIN {X 0,Y 545.08,Z 90.716,A -85,B 0,C 180,E1 -3803.56,E2 -3803.56} C_VEL
LIN {X 0,Y 545.078,Z 90.709,A -85,B 0,C 180,E1 -3806.001,E2 -3806.001} C_VEL
LIN {X 0,Y 545.074,Z 90.709,A -85,B 0,C 180,E1 -3808.746,E2 -3808.746} C_VEL
LIN {X 0,Y 545.057,Z 90.713,A -85,B 0,C 180,E1 -3811.679,E2 -3811.679} C_VEL
LIN {X 0,Y 545.059,Z 90.711,A -85,B 0,C 180,E1 -3814.565,E2 -3814.565} C_VEL
LIN {X 0,Y 545.062,Z 90.716,A -85,B 0,C 180,E1 -3816.993,E2 -3816.993} C_VEL
LIN {X 0,Y 544.353,Z 90.802,A -85,B 0,C 180,E1 -3817.61,E2 -3817.61} C_VEL
LIN {X 0,Y 541.481,Z 91.159,A -85,B 0,C 180,E1 -3818.61,E2 -3818.61} C_VEL
LIN {X 0,Y 539.091,Z 91.457,A -85,B 0,C 180,E1 -3819.416,E2 -3819.416} C_VEL
LIN {X 0,Y 538.084,Z 91.579,A -85,B 0,C 180,E1 -3820.038,E2 -3820.038} C_VEL
LIN {X 0,Y 538.01,Z 91.589,A -85,B 0,C 180,E1 -3820.249,E2 -3820.249} C_VEL
LIN {X 0,Y 538.027,Z 91.594,A -85,B 0,C 180,E1 -3822.988,E2 -3822.988} C_VEL
LIN {X 0,Y 538.02,Z 91.587,A -85,B 0,C 180,E1 -3825.927,E2 -3825.927} C_VEL
LIN {X 0,Y 538.049,Z 91.585,A -85,B 0,C 180,E1 -3829.253,E2 -3829.253} C_VEL
LIN {X 0,Y 537.989,Z 91.593,A -85,B 0,C 180,E1 -3832.122,E2 -3832.122} C_VEL
LIN {X 0,Y 537.996,Z 91.593,A -85,B 0,C 180,E1 -3834.916,E2 -3834.916} C_VEL
LIN {X 0,Y 538.02,Z 91.587,A -85,B 0,C 180,E1 -3837.618,E2 -3837.618} C_VEL
LIN {X 0,Y 538.015,Z 91.596,A -85,B 0,C 180,E1 -3840.239,E2 -3840.239} C_VEL
LIN {X 0,Y 538.014,Z 91.589,A -85,B 0,C 180,E1 -3842.794,E2 -3842.794} C_VEL
LIN {X 0,Y 538.018,Z 91.587,A -85,B 0,C 180,E1 -3845.291,E2 -3845.291} C_VEL
LIN {X 0,Y 538.018,Z 91.596,A -85,B 0,C 180,E1 -3848.042,E2 -3848.042} C_VEL
LIN {X 0,Y 538.083,Z 91.587,A -85,B 0,C 180,E1 -3850.148,E2 -3850.148} C_VEL
LIN {X 0,Y 538.044,Z 91.705,A -85,B 0,C 180,E1 -3853.446,E2 -3853.446} C_VEL
LIN {X 0,Y 539.216,Z 98.867,A -85,B 0,C 180,E1 -3854.688,E2 -3854.688} C_VEL
LIN {X 0,Y 538.811,Z 116.611,A -85,B 0,C 180,E1 -3857.572,E2 -3857.572} C_VEL
LIN {X 0,Y 538.773,Z 120.472,A -85,B 0,C 180,E1 -3858.179,E2 -3858.179} C_VEL
LIN {X 0,Y 540.694,Z 130.72,A -85,B 0,C 180,E1 -3858.385,E2 -3858.385} C_VEL
LIN {X 0,Y 540.115,Z 256.487,A -85,B 0,C 180,E1 -3860.096,E2 -3860.096} C_VEL
LIN {X 0,Y 539.941,Z 271.122,A -85,B 0,C 180,E1 -3860.447,E2 -3860.447} C_VEL
LIN {X 0,Y 539.749,Z 284.433,A -85,B 0,C 180,E1 -3860.916,E2 -3860.916} C_VEL
LIN {X 0,Y 539.403,Z 298.333,A -85,B 0,C 180,E1 -3861.571,E2 -3861.571} C_VEL
LIN {X 0,Y 539.041,Z 311.033,A -85,B 0,C 180,E1 -3862.339,E2 -3862.339} C_VEL
LIN {X 0,Y 538.786,Z 323.234,A -85,B 0,C 180,E1 -3863.258,E2 -3863.258} C_VEL
LIN {X 0,Y 538.479,Z 333.476,A -85,B 0,C 180,E1 -3864.195,E2 -3864.195} C_VEL
LIN {X 0,Y 538.232,Z 343.691,A -85,B 0,C 180,E1 -3865.319,E2 -3865.319} C_VEL
LIN {X 0,Y 537.988,Z 352.149,A -85,B 0,C 180,E1 -3866.443,E2 -3866.443} C_VEL
LIN {X 0,Y 537.704,Z 360.291,A -85,B 0,C 180,E1 -3867.753,E2 -3867.753} C_VEL
LIN {X 0,Y 537.717,Z 365.97,A -85,B 0,C 180,E1 -3868.877,E2 -3868.877} C_VEL
LIN {X 0,Y 537.555,Z 370.668,A -85,B 0,C 180,E1 -3870,E2 -3870} C_VEL
LIN {X 0,Y 537.487,Z 375.544,A -85,B 0,C 180,E1 -3871.499,E2 -3871.499} C_VEL
LIN {X 0,Y 537.573,Z 378.946,A -85,B 0,C 180,E1 -3872.998,E2 -3872.998} C_VEL
LIN {X 0,Y 537.493,Z 380.984,A -85,B 0,C 180,E1 -3874.5,E2 -3874.5} C_VEL
LIN {X 0,Y 537.526,Z 381.689,A -85,B 0,C 180,E1 -3876.004,E2 -3876.004} C_VEL
LIN {X 0,Y 537.517,Z 381.062,A -85,B 0,C 180,E1 -3877.513,E2 -3877.513} C_VEL
LIN {X 0,Y 537.473,Z 379.071,A -85,B 0,C 180,E1 -3879.028,E2 -3879.028} C_VEL
LIN {X 0,Y 537.557,Z 375.665,A -85,B 0,C 180,E1 -3880.547,E2 -3880.547} C_VEL
LIN {X 0,Y 537.614,Z 370.732,A -85,B 0,C 180,E1 -3882.073,E2 -3882.073} C_VEL
LIN {X 0,Y 537.7,Z 365.933,A -85,B 0,C 180,E1 -3883.223,E2 -3883.223} C_VEL
LIN {X 0,Y 537.875,Z 358.389,A -85,B 0,C 180,E1 -3884.662,E2 -3884.662} C_VEL
LIN {X 0,Y 538.028,Z 350.21,A -85,B 0,C 180,E1 -3885.921,E2 -3885.921} C_VEL
LIN {X 0,Y 538.291,Z 341.032,A -85,B 0,C 180,E1 -3887.083,E2 -3887.083} C_VEL
LIN {X 0,Y 538.572,Z 329.844,A -85,B 0,C 180,E1 -3888.251,E2 -3888.251} C_VEL
LIN {X 0,Y 538.897,Z 318.346,A -85,B 0,C 180,E1 -3889.226,E2 -3889.226} C_VEL
LIN {X 0,Y 539.205,Z 305.823,A -85,B 0,C 180,E1 -3890.088,E2 -3890.088} C_VEL
LIN {X 0,Y 539.52,Z 293.022,A -85,B 0,C 180,E1 -3890.792,E2 -3890.792} C_VEL
LIN {X 0,Y 539.82,Z 279.109,A -85,B 0,C 180,E1 -3891.379,E2 -3891.379} C_VEL
LIN {X 0,Y 539.998,Z 265.459,A -85,B 0,C 180,E1 -3891.798,E2 -3891.798} C_VEL
LIN {X 0,Y 540.138,Z 251.896,A -85,B 0,C 180,E1 -3892.068,E2 -3892.068} C_VEL
LIN {X 0,Y 540.631,Z 129.71,A -85,B 0,C 180,E1 -3893.721,E2 -3893.721} C_VEL
LIN {X 0,Y 538.754,Z 120.283,A -85,B 0,C 180,E1 -3893.93,E2 -3893.93} C_VEL
LIN {X 0,Y 539.102,Z 104.297,A -85,B 0,C 180,E1 -3896.519,E2 -3896.519} C_VEL
LIN {X 0,Y 539.052,Z 97.114,A -85,B 0,C 180,E1 -3897.704,E2 -3897.704} C_VEL
LIN {X 0,Y 537.985,Z 91.598,A -85,B 0,C 180,E1 -3898.691,E2 -3898.691} C_VEL
LIN {X 0,Y 537.99,Z 91.596,A -85,B 0,C 180,E1 -3901.503,E2 -3901.503} C_VEL
LIN {X 0,Y 537.991,Z 91.597,A -85,B 0,C 180,E1 -3904.175,E2 -3904.175} C_VEL
LIN {X 0,Y 537.962,Z 91.595,A -85,B 0,C 180,E1 -3907.163,E2 -3907.163} C_VEL
LIN {X 0,Y 537.97,Z 91.602,A -85,B 0,C 180,E1 -3909.802,E2 -3909.802} C_VEL
LIN {X 0,Y 537.96,Z 91.595,A -85,B 0,C 180,E1 -3912.792,E2 -3912.792} C_VEL
LIN {X 0,Y 537.99,Z 91.594,A -85,B 0,C 180,E1 -3915.136,E2 -3915.136} C_VEL
LIN {X 0,Y 537.985,Z 91.592,A -85,B 0,C 180,E1 -3918.222,E2 -3918.222} C_VEL
LIN {X 0,Y 538.005,Z 91.591,A -85,B 0,C 180,E1 -3921.168,E2 -3921.168} C_VEL
LIN {X 0,Y 537.988,Z 91.591,A -85,B 0,C 180,E1 -3924.09,E2 -3924.09} C_VEL
LIN {X 0,Y 538.032,Z 91.589,A -85,B 0,C 180,E1 -3926.727,E2 -3926.727} C_VEL
LIN {X 0,Y 538.004,Z 91.59,A -85,B 0,C 180,E1 -3929.561,E2 -3929.561} C_VEL
LIN {X 0,Y 538.01,Z 91.594,A -85,B 0,C 180,E1 -3932.658,E2 -3932.658} C_VEL
LIN {X 0,Y 537.982,Z 91.595,A -85,B 0,C 180,E1 -3935.289,E2 -3935.289} C_VEL
LIN {X 0,Y 538.015,Z 91.586,A -85,B 0,C 180,E1 -3938.042,E2 -3938.042} C_VEL
LIN {X 0,Y 538.082,Z 91.582,A -85,B 0,C 180,E1 -3940.148,E2 -3940.148} C_VEL
LIN {X 0,Y 538.002,Z 91.59,A -85,B 0,C 180,E1 -3943.298,E2 -3943.298} C_VEL
LIN {X 0,Y 538.04,Z 91.584,A -85,B 0,C 180,E1 -3945.63,E2 -3945.63} C_VEL
LIN {X 0,Y 538.077,Z 91.584,A -85,B 0,C 180,E1 -3948.701,E2 -3948.701} C_VEL
LIN {X 0,Y 538.061,Z 91.581,A -85,B 0,C 180,E1 -3951.739,E2 -3951.739} C_VEL
LIN {X 0,Y 538.154,Z 91.571,A -85,B 0,C 180,E1 -3954.755,E2 -3954.755} C_VEL
LIN {X 0,Y 538.167,Z 91.573,A -85,B 0,C 180,E1 -3957.755,E2 -3957.755} C_VEL
LIN {X 0,Y 538.18,Z 91.565,A -85,B 0,C 180,E1 -3960.748,E2 -3960.748} C_VEL
LIN {X 0,Y 538.133,Z 91.573,A -85,B 0,C 180,E1 -3962.994,E2 -3962.994} C_VEL
LIN {X 0,Y 538.093,Z 91.58,A -85,B 0,C 180,E1 -3965.998,E2 -3965.998} C_VEL
LIN {X 0,Y 538.059,Z 91.584,A -85,B 0,C 180,E1 -3969.018,E2 -3969.018} C_VEL
LIN {X 0,Y 538.067,Z 91.582,A -85,B 0,C 180,E1 -3972.063,E2 -3972.063} C_VEL
LIN {X 0,Y 538.043,Z 91.59,A -85,B 0,C 180,E1 -3975.144,E2 -3975.144} C_VEL
LIN {X 0,Y 538.029,Z 91.586,A -85,B 0,C 180,E1 -3978.27,E2 -3978.27} C_VEL
LIN {X 0,Y 538.038,Z 91.585,A -85,B 0,C 180,E1 -3980.651,E2 -3980.651} C_VEL
LIN {X 0,Y 538.003,Z 91.588,A -85,B 0,C 180,E1 -3983.888,E2 -3983.888} C_VEL
LIN {X 0,Y 538.043,Z 91.585,A -85,B 0,C 180,E1 -3986.367,E2 -3986.367} C_VEL
LIN {X 0,Y 538.032,Z 91.592,A -85,B 0,C 180,E1 -3988.933,E2 -3988.933} C_VEL
LIN {X 0,Y 538.016,Z 91.587,A -85,B 0,C 180,E1 -3991.888,E2 -3991.888} C_VEL
LIN {X 0,Y 538.023,Z 91.596,A -85,B 0,C 180,E1 -3994.619,E2 -3994.619} C_VEL
LIN {X 0,Y 538.004,Z 91.591,A -85,B 0,C 180,E1 -3997.17,E2 -3997.17} C_VEL
LIN {X 0,Y 538.023,Z 91.583,A -85,B 0,C 180,E1 -3999.797,E2 -3999.797} C_VEL
LIN {X 0,Y 538.02,Z 91.59,A -85,B 0,C 180,E1 -4002.786,E2 -4002.786} C_VEL
LIN {X 0,Y 538.008,Z 91.588,A -85,B 0,C 180,E1 -4005.138,E2 -4005.138} C_VEL
LIN {X 0,Y 538.035,Z 91.594,A -85,B 0,C 180,E1 -4008.227,E2 -4008.227} C_VEL
LIN {X 0,Y 538.017,Z 91.587,A -85,B 0,C 180,E1 -4011.17,E2 -4011.17} C_VEL
LIN {X 0,Y 537.995,Z 91.597,A -85,B 0,C 180,E1 -4014.089,E2 -4014.089} C_VEL
LIN {X 0,Y 538.032,Z 91.584,A -85,B 0,C 180,E1 -4016.727,E2 -4016.727} C_VEL
LIN {X 0,Y 538.028,Z 91.593,A -85,B 0,C 180,E1 -4019.556,E2 -4019.556} C_VEL
LIN {X 0,Y 538.046,Z 91.592,A -85,B 0,C 180,E1 -4021.95,E2 -4021.95} C_VEL
LIN {X 0,Y 538.076,Z 91.63,A -85,B 0,C 180,E1 -4024.726,E2 -4024.726} C_VEL
LIN {X 0,Y 539.602,Z 99.215,A -85,B 0,C 180,E1 -4025.912,E2 -4025.912} C_VEL
LIN {X 0,Y 539.528,Z 109.488,A -85,B 0,C 180,E1 -4027.396,E2 -4027.396} C_VEL
LIN {X 0,Y 539.028,Z 130.583,A -85,B 0,C 180,E1 -4030.383,E2 -4030.383} C_VEL
LIN {X 0,Y 538.793,Z 143.014,A -85,B 0,C 180,E1 -4032.121,E2 -4032.121} C_VEL
LIN {X 0,Y 540.654,Z 154.828,A -85,B 0,C 180,E1 -4032.345,E2 -4032.345} C_VEL
LIN {X 0,Y 540.056,Z 281.26,A -85,B 0,C 180,E1 -4034.068,E2 -4034.068} C_VEL
LIN {X 0,Y 539.848,Z 295.7,A -85,B 0,C 180,E1 -4034.422,E2 -4034.422} C_VEL
LIN {X 0,Y 539.641,Z 309.148,A -85,B 0,C 180,E1 -4034.902,E2 -4034.902} C_VEL
LIN {X 0,Y 539.339,Z 321.348,A -85,B 0,C 180,E1 -4035.473,E2 -4035.473} C_VEL
LIN {X 0,Y 538.988,Z 334.186,A -85,B 0,C 180,E1 -4036.233,E2 -4036.233} C_VEL
LIN {X 0,Y 538.677,Z 345.861,A -85,B 0,C 180,E1 -4037.09,E2 -4037.09} C_VEL
LIN {X 0,Y 538.453,Z 357.003,A -85,B 0,C 180,E1 -4038.085,E2 -4038.085} C_VEL
LIN {X 0,Y 538.219,Z 366.349,A -85,B 0,C 180,E1 -4039.086,E2 -4039.086} C_VEL
LIN {X 0,Y 537.96,Z 375.239,A -85,B 0,C 180,E1 -4040.222,E2 -4040.222} C_VEL
LIN {X 0,Y 537.815,Z 383.761,A -85,B 0,C 180,E1 -4041.546,E2 -4041.546} C_VEL
LIN {X 0,Y 537.658,Z 390.628,A -85,B 0,C 180,E1 -4042.867,E2 -4042.867} C_VEL
LIN {X 0,Y 537.634,Z 396.763,A -85,B 0,C 180,E1 -4044.374,E2 -4044.374} C_VEL
LIN {X 0,Y 537.548,Z 400.266,A -85,B 0,C 180,E1 -4045.501,E2 -4045.501} C_VEL
LIN {X 0,Y 537.546,Z 403.676,A -85,B 0,C 180,E1 -4047.002,E2 -4047.002} C_VEL
LIN {X 0,Y 537.447,Z 405.691,A -85,B 0,C 180,E1 -4048.501,E2 -4048.501} C_VEL
LIN {X 0,Y 537.441,Z 406.36,A -85,B 0,C 180,E1 -4050,E2 -4050} C_VEL
LIN {X 0,Y 537.447,Z 405.694,A -85,B 0,C 180,E1 -4051.499,E2 -4051.499} C_VEL
LIN {X 0,Y 537.546,Z 403.682,A -85,B 0,C 180,E1 -4052.998,E2 -4052.998} C_VEL
LIN {X 0,Y 537.548,Z 400.272,A -85,B 0,C 180,E1 -4054.499,E2 -4054.499} C_VEL
LIN {X 0,Y 537.631,Z 395.365,A -85,B 0,C 180,E1 -4056.003,E2 -4056.003} C_VEL
LIN {X 0,Y 537.658,Z 390.632,A -85,B 0,C 180,E1 -4057.133,E2 -4057.133} C_VEL
LIN {X 0,Y 537.815,Z 383.769,A -85,B 0,C 180,E1 -4058.454,E2 -4058.454} C_VEL
LIN {X 0,Y 537.96,Z 375.247,A -85,B 0,C 180,E1 -4059.778,E2 -4059.778} C_VEL
LIN {X 0,Y 538.22,Z 366.359,A -85,B 0,C 180,E1 -4060.914,E2 -4060.914} C_VEL
LIN {X 0,Y 538.453,Z 355.592,A -85,B 0,C 180,E1 -4062.054,E2 -4062.054} C_VEL
LIN {X 0,Y 538.749,Z 344.699,A -85,B 0,C 180,E1 -4063.004,E2 -4063.004} C_VEL
LIN {X 0,Y 539.046,Z 332.777,A -85,B 0,C 180,E1 -4063.861,E2 -4063.861} C_VEL
LIN {X 0,Y 539.371,Z 319.586,A -85,B 0,C 180,E1 -4064.623,E2 -4064.623} C_VEL
LIN {X 0,Y 539.715,Z 307.459,A -85,B 0,C 180,E1 -4065.168,E2 -4065.168} C_VEL
LIN {X 0,Y 539.88,Z 293.149,A -85,B 0,C 180,E1 -4065.655,E2 -4065.655} C_VEL
LIN {X 0,Y 540.077,Z 278.516,A -85,B 0,C 180,E1 -4065.98,E2 -4065.98} C_VEL
LIN {X 0,Y 540.654,Z 153.782,A -85,B 0,C 180,E1 -4067.669,E2 -4067.669} C_VEL
LIN {X 0,Y 538.803,Z 142.99,A -85,B 0,C 180,E1 -4067.885,E2 -4067.885} C_VEL
LIN {X 0,Y 539.219,Z 122.194,A -85,B 0,C 180,E1 -4070.803,E2 -4070.803} C_VEL
LIN {X 0,Y 539.745,Z 101.14,A -85,B 0,C 180,E1 -4073.806,E2 -4073.806} C_VEL
LIN {X 0,Y 538.918,Z 95.494,A -85,B 0,C 180,E1 -4074.665,E2 -4074.665} C_VEL
LIN {X 0,Y 538.069,Z 91.587,A -85,B 0,C 180,E1 -4075.274,E2 -4075.274} C_VEL
LIN {X 0,Y 538.045,Z 91.59,A -85,B 0,C 180,E1 -4078.049,E2 -4078.049} C_VEL
LIN {X 0,Y 538.021,Z 91.592,A -85,B 0,C 180,E1 -4080.627,E2 -4080.627} C_VEL
LIN {X 0,Y 538.046,Z 91.584,A -85,B 0,C 180,E1 -4083.283,E2 -4083.283} C_VEL
LIN {X 0,Y 537.994,Z 91.598,A -85,B 0,C 180,E1 -4086.004,E2 -4086.004} C_VEL
LIN {X 0,Y 538.015,Z 91.588,A -85,B 0,C 180,E1 -4088.83,E2 -4088.83} C_VEL
LIN {X 0,Y 538.039,Z 91.592,A -85,B 0,C 180,E1 -4091.772,E2 -4091.772} C_VEL
LIN {X 0,Y 538.032,Z 91.585,A -85,B 0,C 180,E1 -4094.859,E2 -4094.859} C_VEL
LIN {X 0,Y 538.034,Z 91.588,A -85,B 0,C 180,E1 -4098.121,E2 -4098.121} C_VEL
LIN {X 0,Y 538.032,Z 91.586,A -85,B 0,C 180,E1 -4100.415,E2 -4100.415} C_VEL
LIN {X 0,Y 538.023,Z 91.589,A -85,B 0,C 180,E1 -4103.067,E2 -4103.067} C_VEL
LIN {X 0,Y 538.019,Z 91.59,A -85,B 0,C 180,E1 -4105.827,E2 -4105.827} C_VEL
LIN {X 0,Y 538.009,Z 91.588,A -85,B 0,C 180,E1 -4108.499,E2 -4108.499} C_VEL
LIN {X 0,Y 538.059,Z 91.589,A -85,B 0,C 180,E1 -4111.1,E2 -4111.1} C_VEL
LIN {X 0,Y 538.041,Z 91.587,A -85,B 0,C 180,E1 -4113.633,E2 -4113.633} C_VEL
LIN {X 0,Y 538.006,Z 91.589,A -85,B 0,C 180,E1 -4116.122,E2 -4116.122} C_VEL
LIN {X 0,Y 538.036,Z 91.589,A -85,B 0,C 180,E1 -4119.349,E2 -4119.349} C_VEL
LIN {X 0,Y 538.054,Z 91.586,A -85,B 0,C 180,E1 -4122.517,E2 -4122.517} C_VEL
LIN {X 0,Y 538.064,Z 91.582,A -85,B 0,C 180,E1 -4125.631,E2 -4125.631} C_VEL
LIN {X 0,Y 538.076,Z 91.589,A -85,B 0,C 180,E1 -4128.702,E2 -4128.702} C_VEL
LIN {X 0,Y 538.084,Z 91.579,A -85,B 0,C 180,E1 -4131.74,E2 -4131.74} C_VEL
LIN {X 0,Y 538.159,Z 91.575,A -85,B 0,C 180,E1 -4134.755,E2 -4134.755} C_VEL
LIN {X 0,Y 538.166,Z 91.57,A -85,B 0,C 180,E1 -4137.755,E2 -4137.755} C_VEL
LIN {X 0,Y 538.181,Z 91.569,A -85,B 0,C 180,E1 -4140.748,E2 -4140.748} C_VEL
LIN {X 0,Y 538.136,Z 91.573,A -85,B 0,C 180,E1 -4142.995,E2 -4142.995} C_VEL
LIN {X 0,Y 538.113,Z 91.583,A -85,B 0,C 180,E1 -4145.998,E2 -4145.998} C_VEL
LIN {X 0,Y 538.068,Z 91.581,A -85,B 0,C 180,E1 -4149.018,E2 -4149.018} C_VEL
LIN {X 0,Y 538.083,Z 91.586,A -85,B 0,C 180,E1 -4152.063,E2 -4152.063} C_VEL
LIN {X 0,Y 538.044,Z 91.585,A -85,B 0,C 180,E1 -4155.144,E2 -4155.144} C_VEL
LIN {X 0,Y 538.015,Z 91.589,A -85,B 0,C 180,E1 -4158.271,E2 -4158.271} C_VEL
LIN {X 0,Y 538.038,Z 91.585,A -85,B 0,C 180,E1 -4160.652,E2 -4160.652} C_VEL
LIN {X 0,Y 538.003,Z 91.593,A -85,B 0,C 180,E1 -4163.889,E2 -4163.889} C_VEL
LIN {X 0,Y 538.041,Z 91.584,A -85,B 0,C 180,E1 -4166.367,E2 -4166.367} C_VEL
LIN {X 0,Y 538.029,Z 91.589,A -85,B 0,C 180,E1 -4168.934,E2 -4168.934} C_VEL
LIN {X 0,Y 538.009,Z 91.589,A -85,B 0,C 180,E1 -4171.887,E2 -4171.887} C_VEL
LIN {X 0,Y 538.009,Z 91.59,A -85,B 0,C 180,E1 -4174.617,E2 -4174.617} C_VEL
LIN {X 0,Y 538.004,Z 91.597,A -85,B 0,C 180,E1 -4177.17,E2 -4177.17} C_VEL
LIN {X 0,Y 538.01,Z 91.589,A -85,B 0,C 180,E1 -4180.249,E2 -4180.249} C_VEL
LIN {X 0,Y 537.366,Z 91.676,A -85,B 0,C 180,E1 -4180.874,E2 -4180.874} C_VEL
LIN {X 0,Y 534.516,Z 92.03,A -85,B 0,C 180,E1 -4181.889,E2 -4181.889} C_VEL
LIN {X 0,Y 532.089,Z 92.332,A -85,B 0,C 180,E1 -4182.706,E2 -4182.706} C_VEL
LIN {X 0,Y 531.041,Z 92.459,A -85,B 0,C 180,E1 -4183.337,E2 -4183.337} C_VEL
LIN {X 0,Y 530.953,Z 92.468,A -85,B 0,C 180,E1 -4183.551,E2 -4183.551} C_VEL
LIN {X 0,Y 530.945,Z 92.473,A -85,B 0,C 180,E1 -4186.504,E2 -4186.504} C_VEL
LIN {X 0,Y 530.981,Z 92.464,A -85,B 0,C 180,E1 -4189.567,E2 -4189.567} C_VEL
LIN {X 0,Y 530.966,Z 92.475,A -85,B 0,C 180,E1 -4192.578,E2 -4192.578} C_VEL
LIN {X 0,Y 530.982,Z 92.464,A -85,B 0,C 180,E1 -4195.31,E2 -4195.31} C_VEL
LIN {X 0,Y 530.968,Z 92.469,A -85,B 0,C 180,E1 -4198.032,E2 -4198.032} C_VEL
LIN {X 0,Y 530.99,Z 92.464,A -85,B 0,C 180,E1 -4200.875,E2 -4200.875} C_VEL
LIN {X 0,Y 530.977,Z 92.472,A -85,B 0,C 180,E1 -4204.101,E2 -4204.101} C_VEL
LIN {X 0,Y 530.955,Z 92.469,A -85,B 0,C 180,E1 -4206.603,E2 -4206.603} C_VEL
LIN {X 0,Y 531.001,Z 92.463,A -85,B 0,C 180,E1 -4209.062,E2 -4209.062} C_VEL
LIN {X 0,Y 530.977,Z 92.47,A -85,B 0,C 180,E1 -4211.478,E2 -4211.478} C_VEL
LIN {X 0,Y 531.006,Z 92.651,A -85,B 0,C 180,E1 -4213.27,E2 -4213.27} C_VEL
LIN {X 0,Y 532.299,Z 99.879,A -85,B 0,C 180,E1 -4214.543,E2 -4214.543} C_VEL
LIN {X 0,Y 531.882,Z 117.283,A -85,B 0,C 180,E1 -4217.407,E2 -4217.407} C_VEL
LIN {X 0,Y 531.818,Z 120.653,A -85,B 0,C 180,E1 -4217.937,E2 -4217.937} C_VEL
LIN {X 0,Y 533.925,Z 130.95,A -85,B 0,C 180,E1 -4218.155,E2 -4218.155} C_VEL
LIN {X 0,Y 533.303,Z 257.131,A -85,B 0,C 180,E1 -4219.896,E2 -4219.896} C_VEL
LIN {X 0,Y 533.112,Z 271.57,A -85,B 0,C 180,E1 -4220.252,E2 -4220.252} C_VEL
LIN {X 0,Y 532.892,Z 285.361,A -85,B 0,C 180,E1 -4220.751,E2 -4220.751} C_VEL
LIN {X 0,Y 532.532,Z 298.231,A -85,B 0,C 180,E1 -4221.366,E2 -4221.366} C_VEL
LIN {X 0,Y 532.141,Z 310.997,A -85,B 0,C 180,E1 -4222.145,E2 -4222.145} C_VEL
LIN {X 0,Y 531.829,Z 323.355,A -85,B 0,C 180,E1 -4223.085,E2 -4223.085} C_VEL
LIN {X 0,Y 531.489,Z 334.453,A -85,B 0,C 180,E1 -4224.118,E2 -4224.118} C_VEL
LIN {X 0,Y 531.212,Z 344.51,A -85,B 0,C 180,E1 -4225.257,E2 -4225.257} C_VEL
LIN {X 0,Y 530.944,Z 352.867,A -85,B 0,C 180,E1 -4226.395,E2 -4226.395} C_VEL
LIN {X 0,Y 530.635,Z 360.878,A -85,B 0,C 180,E1 -4227.723,E2 -4227.723} C_VEL
LIN {X 0,Y 530.65,Z 366.512,A -85,B 0,C 180,E1 -4228.862,E2 -4228.862} C_VEL
LIN {X 0,Y 530.469,Z 371.13,A -85,B 0,C 180,E1 -4230,E2 -4230} C_VEL
LIN {X 0,Y 530.394,Z 375.931,A -85,B 0,C 180,E1 -4231.519,E2 -4231.519} C_VEL
LIN {X 0,Y 530.475,Z 379.263,A -85,B 0,C 180,E1 -4233.038,E2 -4233.038} C_VEL
LIN {X 0,Y 530.395,Z 381.228,A -85,B 0,C 180,E1 -4234.56,E2 -4234.56} C_VEL
LIN {X 0,Y 530.444,Z 381.852,A -85,B 0,C 180,E1 -4236.085,E2 -4236.085} C_VEL
LIN {X 0,Y 530.427,Z 381.142,A -85,B 0,C 180,E1 -4237.614,E2 -4237.614} C_VEL
LIN {X 0,Y 530.38,Z 379.08,A -85,B 0,C 180,E1 -4239.15,E2 -4239.15} C_VEL
LIN {X 0,Y 530.491,Z 375.601,A -85,B 0,C 180,E1 -4240.689,E2 -4240.689} C_VEL
LIN {X 0,Y 530.513,Z 372.026,A -85,B 0,C 180,E1 -4241.849,E2 -4241.849} C_VEL
LIN {X 0,Y 530.611,Z 367.456,A -85,B 0,C 180,E1 -4243.013,E2 -4243.013} C_VEL
LIN {X 0,Y 530.732,Z 360.827,A -85,B 0,C 180,E1 -4244.376,E2 -4244.376} C_VEL
LIN {X 0,Y 530.942,Z 352.538,A -85,B 0,C 180,E1 -4245.745,E2 -4245.745} C_VEL
LIN {X 0,Y 531.193,Z 343.801,A -85,B 0,C 180,E1 -4246.922,E2 -4246.922} C_VEL
LIN {X 0,Y 531.522,Z 333.147,A -85,B 0,C 180,E1 -4248.103,E2 -4248.103} C_VEL
LIN {X 0,Y 531.853,Z 322.342,A -85,B 0,C 180,E1 -4249.09,E2 -4249.09} C_VEL
LIN {X 0,Y 532.137,Z 310.472,A -85,B 0,C 180,E1 -4249.983,E2 -4249.983} C_VEL
LIN {X 0,Y 532.535,Z 298.33,A -85,B 0,C 180,E1 -4250.719,E2 -4250.719} C_VEL
LIN {X 0,Y 532.898,Z 284.771,A -85,B 0,C 180,E1 -4251.366,E2 -4251.366} C_VEL
LIN {X 0,Y 533.099,Z 270.763,A -85,B 0,C 180,E1 -4251.866,E2 -4251.866} C_VEL
LIN {X 0,Y 533.289,Z 256.068,A -85,B 0,C 180,E1 -4252.214,E2 -4252.214} C_VEL
LIN {X 0,Y 533.838,Z 130.322,A -85,B 0,C 180,E1 -4253.947,E2 -4253.947} C_VEL
LIN {X 0,Y 531.829,Z 120.495,A -85,B 0,C 180,E1 -4254.163,E2 -4254.163} C_VEL
LIN {X 0,Y 532.181,Z 105.145,A -85,B 0,C 180,E1 -4256.68,E2 -4256.68} C_VEL
LIN {X 0,Y 532.147,Z 98.655,A -85,B 0,C 180,E1 -4257.765,E2 -4257.765} C_VEL
LIN {X 0,Y 530.938,Z 92.475,A -85,B 0,C 180,E1 -4258.907,E2 -4258.907} C_VEL
LIN {X 0,Y 530.953,Z 92.476,A -85,B 0,C 180,E1 -4261.969,E2 -4261.969} C_VEL
LIN {X 0,Y 530.954,Z 92.468,A -85,B 0,C 180,E1 -4264.848,E2 -4264.848} C_VEL
LIN {X 0,Y 530.927,Z 92.474,A -85,B 0,C 180,E1 -4267.511,E2 -4267.511} C_VEL
LIN {X 0,Y 530.908,Z 92.475,A -85,B 0,C 180,E1 -4270.44,E2 -4270.44} C_VEL
LIN {X 0,Y 530.92,Z 92.479,A -85,B 0,C 180,E1 -4273.499,E2 -4273.499} C_VEL
LIN {X 0,Y 530.965,Z 92.47,A -85,B 0,C 180,E1 -4275.624,E2 -4275.624} C_VEL
LIN {X 0,Y 530.936,Z 92.473,A -85,B 0,C 180,E1 -4278.983,E2 -4278.983} C_VEL
LIN {X 0,Y 530.949,Z 92.475,A -85,B 0,C 180,E1 -4281.528,E2 -4281.528} C_VEL
LIN {X 0,Y 530.948,Z 92.467,A -85,B 0,C 180,E1 -4284.379,E2 -4284.379} C_VEL
LIN {X 0,Y 530.967,Z 92.473,A -85,B 0,C 180,E1 -4287.133,E2 -4287.133} C_VEL
LIN {X 0,Y 530.949,Z 92.467,A -85,B 0,C 180,E1 -4289.801,E2 -4289.801} C_VEL
LIN {X 0,Y 530.965,Z 92.469,A -85,B 0,C 180,E1 -4292.478,E2 -4292.478} C_VEL
LIN {X 0,Y 530.949,Z 92.476,A -85,B 0,C 180,E1 -4294.939,E2 -4294.939} C_VEL
LIN {X 0,Y 530.977,Z 92.462,A -85,B 0,C 180,E1 -4297.898,E2 -4297.898} C_VEL
LIN {X 0,Y 530.983,Z 92.47,A -85,B 0,C 180,E1 -4300.677,E2 -4300.677} C_VEL
LIN {X 0,Y 530.964,Z 92.469,A -85,B 0,C 180,E1 -4303.07,E2 -4303.07} C_VEL
LIN {X 0,Y 531,Z 92.461,A -85,B 0,C 180,E1 -4305.435,E2 -4305.435} C_VEL
LIN {X 0,Y 531.035,Z 92.464,A -85,B 0,C 180,E1 -4308.55,E2 -4308.55} C_VEL
LIN {X 0,Y 531.036,Z 92.455,A -85,B 0,C 180,E1 -4311.629,E2 -4311.629} C_VEL
LIN {X 0,Y 531.114,Z 92.448,A -85,B 0,C 180,E1 -4314.685,E2 -4314.685} C_VEL
LIN {X 0,Y 531.138,Z 92.447,A -85,B 0,C 180,E1 -4317.725,E2 -4317.725} C_VEL
LIN {X 0,Y 531.15,Z 92.441,A -85,B 0,C 180,E1 -4320.758,E2 -4320.758} C_VEL
LIN {X 0,Y 531.1,Z 92.449,A -85,B 0,C 180,E1 -4323.034,E2 -4323.034} C_VEL
LIN {X 0,Y 531.051,Z 92.456,A -85,B 0,C 180,E1 -4326.077,E2 -4326.077} C_VEL
LIN {X 0,Y 531.02,Z 92.462,A -85,B 0,C 180,E1 -4329.138,E2 -4329.138} C_VEL
LIN {X 0,Y 531.031,Z 92.457,A -85,B 0,C 180,E1 -4332.225,E2 -4332.225} C_VEL
LIN {X 0,Y 530.994,Z 92.469,A -85,B 0,C 180,E1 -4335.35,E2 -4335.35} C_VEL
LIN {X 0,Y 530.988,Z 92.463,A -85,B 0,C 180,E1 -4338.521,E2 -4338.521} C_VEL
LIN {X 0,Y 530.999,Z 92.465,A -85,B 0,C 180,E1 -4340.938,E2 -4340.938} C_VEL
LIN {X 0,Y 530.972,Z 92.464,A -85,B 0,C 180,E1 -4344.225,E2 -4344.225} C_VEL
LIN {X 0,Y 531.003,Z 92.466,A -85,B 0,C 180,E1 -4346.744,E2 -4346.744} C_VEL
LIN {X 0,Y 530.983,Z 92.466,A -85,B 0,C 180,E1 -4349.322,E2 -4349.322} C_VEL
LIN {X 0,Y 530.972,Z 92.466,A -85,B 0,C 180,E1 -4352.101,E2 -4352.101} C_VEL
LIN {X 0,Y 530.979,Z 92.469,A -85,B 0,C 180,E1 -4354.852,E2 -4354.852} C_VEL
LIN {X 0,Y 530.966,Z 92.466,A -85,B 0,C 180,E1 -4357.508,E2 -4357.508} C_VEL
LIN {X 0,Y 530.982,Z 92.467,A -85,B 0,C 180,E1 -4360.433,E2 -4360.433} C_VEL
LIN {X 0,Y 530.965,Z 92.466,A -85,B 0,C 180,E1 -4363.495,E2 -4363.495} C_VEL
LIN {X 0,Y 530.965,Z 92.471,A -85,B 0,C 180,E1 -4366.505,E2 -4366.505} C_VEL
LIN {X 0,Y 530.985,Z 92.466,A -85,B 0,C 180,E1 -4369.567,E2 -4369.567} C_VEL
LIN {X 0,Y 530.969,Z 92.467,A -85,B 0,C 180,E1 -4372.577,E2 -4372.577} C_VEL
LIN {X 0,Y 530.984,Z 92.464,A -85,B 0,C 180,E1 -4375.31,E2 -4375.31} C_VEL
LIN {X 0,Y 530.968,Z 92.471,A -85,B 0,C 180,E1 -4378.032,E2 -4378.032} C_VEL
LIN {X 0,Y 530.99,Z 92.465,A -85,B 0,C 180,E1 -4380.874,E2 -4380.874} C_VEL
LIN {X 0,Y 531.006,Z 92.468,A -85,B 0,C 180,E1 -4383.256,E2 -4383.256} C_VEL
LIN {X 0,Y 531.06,Z 92.593,A -85,B 0,C 180,E1 -4384.526,E2 -4384.526} C_VEL
LIN {X 0,Y 532.752,Z 100.993,A -85,B 0,C 180,E1 -4385.861,E2 -4385.861} C_VEL
LIN {X 0,Y 532.487,Z 114.995,A -85,B 0,C 180,E1 -4387.904,E2 -4387.904} C_VEL
LIN {X 0,Y 532.009,Z 136.033,A -85,B 0,C 180,E1 -4390.916,E2 -4390.916} C_VEL
LIN {X 0,Y 531.818,Z 142.83,A -85,B 0,C 180,E1 -4391.876,E2 -4391.876} C_VEL
LIN {X 0,Y 533.894,Z 154.903,A -85,B 0,C 180,E1 -4392.118,E2 -4392.118} C_VEL
LIN {X 0,Y 533.237,Z 281.08,A -85,B 0,C 180,E1 -4393.858,E2 -4393.858} C_VEL
LIN {X 0,Y 532.991,Z 295.821,A -85,B 0,C 180,E1 -4394.226,E2 -4394.226} C_VEL
LIN {X 0,Y 532.723,Z 310.106,A -85,B 0,C 180,E1 -4394.75,E2 -4394.75} C_VEL
LIN {X 0,Y 532.397,Z 322.945,A -85,B 0,C 180,E1 -4395.377,E2 -4395.377} C_VEL
LIN {X 0,Y 532.032,Z 335.445,A -85,B 0,C 180,E1 -4396.147,E2 -4396.147} C_VEL
LIN {X 0,Y 531.662,Z 348.045,A -85,B 0,C 180,E1 -4397.111,E2 -4397.111} C_VEL
LIN {X 0,Y 531.394,Z 359.095,A -85,B 0,C 180,E1 -4398.151,E2 -4398.151} C_VEL
LIN {X 0,Y 531.086,Z 369.34,A -85,B 0,C 180,E1 -4399.323,E2 -4399.323} C_VEL
LIN {X 0,Y 530.876,Z 377.703,A -85,B 0,C 180,E1 -4400.475,E2 -4400.475} C_VEL
LIN {X 0,Y 530.694,Z 385.699,A -85,B 0,C 180,E1 -4401.815,E2 -4401.815} C_VEL
LIN {X 0,Y 530.572,Z 392.137,A -85,B 0,C 180,E1 -4403.153,E2 -4403.153} C_VEL
LIN {X 0,Y 530.51,Z 397.845,A -85,B 0,C 180,E1 -4404.679,E2 -4404.679} C_VEL
LIN {X 0,Y 530.496,Z 401.987,A -85,B 0,C 180,E1 -4406.202,E2 -4406.202} C_VEL
LIN {X 0,Y 530.41,Z 404.69,A -85,B 0,C 180,E1 -4407.722,E2 -4407.722} C_VEL
LIN {X 0,Y 530.34,Z 406.03,A -85,B 0,C 180,E1 -4409.241,E2 -4409.241} C_VEL
LIN {X 0,Y 530.34,Z 406.031,A -85,B 0,C 180,E1 -4410.759,E2 -4410.759} C_VEL
LIN {X 0,Y 530.41,Z 404.695,A -85,B 0,C 180,E1 -4412.278,E2 -4412.278} C_VEL
LIN {X 0,Y 530.496,Z 401.995,A -85,B 0,C 180,E1 -4413.798,E2 -4413.798} C_VEL
LIN {X 0,Y 530.511,Z 397.851,A -85,B 0,C 180,E1 -4415.321,E2 -4415.321} C_VEL
LIN {X 0,Y 530.572,Z 392.143,A -85,B 0,C 180,E1 -4416.847,E2 -4416.847} C_VEL
LIN {X 0,Y 530.694,Z 385.708,A -85,B 0,C 180,E1 -4418.184,E2 -4418.184} C_VEL
LIN {X 0,Y 530.876,Z 377.714,A -85,B 0,C 180,E1 -4419.525,E2 -4419.525} C_VEL
LIN {X 0,Y 531.086,Z 369.353,A -85,B 0,C 180,E1 -4420.676,E2 -4420.676} C_VEL
LIN {X 0,Y 531.365,Z 359.252,A -85,B 0,C 180,E1 -4421.834,E2 -4421.834} C_VEL
LIN {X 0,Y 531.703,Z 348.063,A -85,B 0,C 180,E1 -4422.888,E2 -4422.888} C_VEL
LIN {X 0,Y 532.016,Z 335.469,A -85,B 0,C 180,E1 -4423.853,E2 -4423.853} C_VEL
LIN {X 0,Y 532.394,Z 322.969,A -85,B 0,C 180,E1 -4424.623,E2 -4424.623} C_VEL
LIN {X 0,Y 532.738,Z 310.122,A -85,B 0,C 180,E1 -4425.249,E2 -4425.249} C_VEL
LIN {X 0,Y 532.99,Z 296.001,A -85,B 0,C 180,E1 -4425.769,E2 -4425.769} C_VEL
LIN {X 0,Y 533.246,Z 282.253,A -85,B 0,C 180,E1 -4426.117,E2 -4426.117} C_VEL
LIN {X 0,Y 533.416,Z 254.127,A -85,B 0,C 180,E1 -4426.529,E2 -4426.529} C_VEL
LIN {X 0,Y 533.837,Z 154.317,A -85,B 0,C 180,E1 -4427.893,E2 -4427.893} C_VEL
LIN {X 0,Y 531.822,Z 142.839,A -85,B 0,C 180,E1 -4428.126,E2 -4428.126} C_VEL
LIN {X 0,Y 532.316,Z 122.046,A -85,B 0,C 180,E1 -4431.086,E2 -4431.086} C_VEL
LIN {X 0,Y 532.832,Z 102.378,A -85,B 0,C 180,E1 -4433.928,E2 -4433.928} C_VEL
LIN {X 0,Y 531.624,Z 95.276,A -85,B 0,C 180,E1 -4435.026,E2 -4435.026} C_VEL
LIN {X 0,Y 531.035,Z 92.463,A -85,B 0,C 180,E1 -4435.475,E2 -4435.475} C_VEL
LIN {X 0,Y 530.999,Z 92.469,A -85,B 0,C 180,E1 -4438.455,E2 -4438.455} C_VEL
LIN {X 0,Y 530.957,Z 92.469,A -85,B 0,C 180,E1 -4441.079,E2 -4441.079} C_VEL
LIN {X 0,Y 530.987,Z 92.466,A -85,B 0,C 180,E1 -4443.772,E2 -4443.772} C_VEL
LIN {X 0,Y 530.955,Z 92.469,A -85,B 0,C 180,E1 -4446.558,E2 -4446.558} C_VEL
LIN {X 0,Y 530.989,Z 92.465,A -85,B 0,C 180,E1 -4449.443,E2 -4449.443} C_VEL
LIN {X 0,Y 530.98,Z 92.466,A -85,B 0,C 180,E1 -4452.456,E2 -4452.456} C_VEL
LIN {X 0,Y 530.988,Z 92.47,A -85,B 0,C 180,E1 -4455.621,E2 -4455.621} C_VEL
LIN {X 0,Y 530.997,Z 92.462,A -85,B 0,C 180,E1 -4458.565,E2 -4458.565} C_VEL
LIN {X 0,Y 530.956,Z 92.475,A -85,B 0,C 180,E1 -4461.529,E2 -4461.529} C_VEL
LIN {X 0,Y 530.953,Z 92.467,A -85,B 0,C 180,E1 -4464.38,E2 -4464.38} C_VEL
LIN {X 0,Y 530.969,Z 92.47,A -85,B 0,C 180,E1 -4467.134,E2 -4467.134} C_VEL
LIN {X 0,Y 530.969,Z 92.468,A -85,B 0,C 180,E1 -4469.803,E2 -4469.803} C_VEL
LIN {X 0,Y 531.011,Z 92.46,A -85,B 0,C 180,E1 -4472.467,E2 -4472.467} C_VEL
LIN {X 0,Y 531.005,Z 92.467,A -85,B 0,C 180,E1 -4474.942,E2 -4474.942} C_VEL
LIN {X 0,Y 530.97,Z 92.465,A -85,B 0,C 180,E1 -4478.247,E2 -4478.247} C_VEL
LIN {X 0,Y 530.992,Z 92.467,A -85,B 0,C 180,E1 -4480.677,E2 -4480.677} C_VEL
LIN {X 0,Y 530.984,Z 92.469,A -85,B 0,C 180,E1 -4483.071,E2 -4483.071} C_VEL
LIN {X 0,Y 531.019,Z 92.46,A -85,B 0,C 180,E1 -4485.436,E2 -4485.436} C_VEL
LIN {X 0,Y 531.036,Z 92.464,A -85,B 0,C 180,E1 -4488.55,E2 -4488.55} C_VEL
LIN {X 0,Y 531.054,Z 92.455,A -85,B 0,C 180,E1 -4491.63,E2 -4491.63} C_VEL
LIN {X 0,Y 531.118,Z 92.453,A -85,B 0,C 180,E1 -4494.685,E2 -4494.685} C_VEL
LIN {X 0,Y 531.138,Z 92.445,A -85,B 0,C 180,E1 -4497.725,E2 -4497.725} C_VEL
LIN {X 0,Y 531.151,Z 92.445,A -85,B 0,C 180,E1 -4500.758,E2 -4500.758} C_VEL
LIN {X 0,Y 531.103,Z 92.449,A -85,B 0,C 180,E1 -4503.034,E2 -4503.034} C_VEL
LIN {X 0,Y 531.067,Z 92.462,A -85,B 0,C 180,E1 -4506.077,E2 -4506.077} C_VEL
LIN {X 0,Y 531.055,Z 92.459,A -85,B 0,C 180,E1 -4508.371,E2 -4508.371} C_VEL
LIN {X 0,Y 531.051,Z 92.46,A -85,B 0,C 180,E1 -4511.672,E2 -4511.672} C_VEL
LIN {X 0,Y 531.031,Z 92.458,A -85,B 0,C 180,E1 -4514.956,E2 -4514.956} C_VEL
LIN {X 0,Y 530.979,Z 92.473,A -85,B 0,C 180,E1 -4517.724,E2 -4517.724} C_VEL
LIN {X 0,Y 531.024,Z 92.461,A -85,B 0,C 180,E1 -4520.127,E2 -4520.127} C_VEL
LIN {X 0,Y 530.945,Z 92.468,A -85,B 0,C 180,E1 -4522.574,E2 -4522.574} C_VEL
LIN {X 0,Y 530.994,Z 92.465,A -85,B 0,C 180,E1 -4525.058,E2 -4525.058} C_VEL
LIN {X 0,Y 531.013,Z 92.466,A -85,B 0,C 180,E1 -4527.596,E2 -4527.596} C_VEL
LIN {X 0,Y 530.966,Z 92.467,A -85,B 0,C 180,E1 -4530.644,E2 -4530.644} C_VEL
LIN {X 0,Y 530.962,Z 92.471,A -85,B 0,C 180,E1 -4533.5,E2 -4533.5} C_VEL
LIN {X 0,Y 530.945,Z 92.468,A -85,B 0,C 180,E1 -4536.154,E2 -4536.154} C_VEL
LIN {X 0,Y 530.965,Z 92.469,A -85,B 0,C 180,E1 -4538.654,E2 -4538.654} C_VEL
LIN {X 0,Y 530.993,Z 92.464,A -85,B 0,C 180,E1 -4541.436,E2 -4541.436} C_VEL
LIN {X 0,Y 530.953,Z 92.468,A -85,B 0,C 180,E1 -4543.551,E2 -4543.551} C_VEL
LIN {X 0,Y 530.28,Z 92.553,A -85,B 0,C 180,E1 -4544.185,E2 -4544.185} C_VEL
LIN {X 0,Y 527.426,Z 92.916,A -85,B 0,C 180,E1 -4545.213,E2 -4545.213} C_VEL
LIN {X 0,Y 525.018,Z 93.22,A -85,B 0,C 180,E1 -4546.042,E2 -4546.042} C_VEL
LIN {X 0,Y 523.985,Z 93.345,A -85,B 0,C 180,E1 -4546.681,E2 -4546.681} C_VEL
LIN {X 0,Y 523.901,Z 93.352,A -85,B 0,C 180,E1 -4546.898,E2 -4546.898} C_VEL
LIN {X 0,Y 523.95,Z 93.34,A -85,B 0,C 180,E1 -4549.921,E2 -4549.921} C_VEL
LIN {X 0,Y 523.905,Z 93.35,A -85,B 0,C 180,E1 -4552.868,E2 -4552.868} C_VEL
LIN {X 0,Y 523.933,Z 93.342,A -85,B 0,C 180,E1 -4555.71,E2 -4555.71} C_VEL
LIN {X 0,Y 523.923,Z 93.351,A -85,B 0,C 180,E1 -4558.456,E2 -4558.456} C_VEL
LIN {X 0,Y 523.928,Z 93.343,A -85,B 0,C 180,E1 -4561.125,E2 -4561.125} C_VEL
LIN {X 0,Y 523.925,Z 93.349,A -85,B 0,C 180,E1 -4563.994,E2 -4563.994} C_VEL
LIN {X 0,Y 523.914,Z 93.351,A -85,B 0,C 180,E1 -4566.27,E2 -4566.27} C_VEL
LIN {X 0,Y 523.948,Z 93.342,A -85,B 0,C 180,E1 -4568.767,E2 -4568.767} C_VEL
LIN {X 0,Y 523.941,Z 93.345,A -85,B 0,C 180,E1 -4571.221,E2 -4571.221} C_VEL
LIN {X 0,Y 523.963,Z 93.421,A -85,B 0,C 180,E1 -4573.063,E2 -4573.063} C_VEL
LIN {X 0,Y 525.374,Z 101.393,A -85,B 0,C 180,E1 -4574.482,E2 -4574.482} C_VEL
LIN {X 0,Y 524.96,Z 117.948,A -85,B 0,C 180,E1 -4577.238,E2 -4577.238} C_VEL
LIN {X 0,Y 524.925,Z 120.84,A -85,B 0,C 180,E1 -4577.692,E2 -4577.692} C_VEL
LIN {X 0,Y 527.196,Z 132.796,A -85,B 0,C 180,E1 -4577.942,E2 -4577.942} C_VEL
LIN {X 0,Y 526.498,Z 257.727,A -85,B 0,C 180,E1 -4579.691,E2 -4579.691} C_VEL
LIN {X 0,Y 526.284,Z 272.02,A -85,B 0,C 180,E1 -4580.051,E2 -4580.051} C_VEL
LIN {X 0,Y 526.032,Z 286.291,A -85,B 0,C 180,E1 -4580.58,E2 -4580.58} C_VEL
LIN {X 0,Y 525.632,Z 299.86,A -85,B 0,C 180,E1 -4581.252,E2 -4581.252} C_VEL
LIN {X 0,Y 525.211,Z 312.345,A -85,B 0,C 180,E1 -4582.04,E2 -4582.04} C_VEL
LIN {X 0,Y 524.885,Z 324.445,A -85,B 0,C 180,E1 -4582.989,E2 -4582.989} C_VEL
LIN {X 0,Y 524.502,Z 335.391,A -85,B 0,C 180,E1 -4584.04,E2 -4584.04} C_VEL
LIN {X 0,Y 524.194,Z 345.294,A -85,B 0,C 180,E1 -4585.193,E2 -4585.193} C_VEL
LIN {X 0,Y 523.9,Z 353.55,A -85,B 0,C 180,E1 -4586.347,E2 -4586.347} C_VEL
LIN {X 0,Y 523.566,Z 361.464,A -85,B 0,C 180,E1 -4587.692,E2 -4587.692} C_VEL
LIN {X 0,Y 523.585,Z 367.039,A -85,B 0,C 180,E1 -4588.846,E2 -4588.846} C_VEL
LIN {X 0,Y 523.418,Z 372.911,A -85,B 0,C 180,E1 -4590.385,E2 -4590.385} C_VEL
LIN {X 0,Y 523.305,Z 376.318,A -85,B 0,C 180,E1 -4591.539,E2 -4591.539} C_VEL
LIN {X 0,Y 523.382,Z 379.571,A -85,B 0,C 180,E1 -4593.079,E2 -4593.079} C_VEL
LIN {X 0,Y 523.303,Z 381.451,A -85,B 0,C 180,E1 -4594.622,E2 -4594.622} C_VEL
LIN {X 0,Y 523.367,Z 381.998,A -85,B 0,C 180,E1 -4596.167,E2 -4596.167} C_VEL
LIN {X 0,Y 523.329,Z 381.22,A -85,B 0,C 180,E1 -4597.718,E2 -4597.718} C_VEL
LIN {X 0,Y 523.289,Z 379.088,A -85,B 0,C 180,E1 -4599.275,E2 -4599.275} C_VEL
LIN {X 0,Y 523.432,Z 375.536,A -85,B 0,C 180,E1 -4600.835,E2 -4600.835} C_VEL
LIN {X 0,Y 523.474,Z 370.445,A -85,B 0,C 180,E1 -4602.405,E2 -4602.405} C_VEL
LIN {X 0,Y 523.604,Z 365.478,A -85,B 0,C 180,E1 -4603.585,E2 -4603.585} C_VEL
LIN {X 0,Y 523.778,Z 358.333,A -85,B 0,C 180,E1 -4604.963,E2 -4604.963} C_VEL
LIN {X 0,Y 523.98,Z 350.736,A -85,B 0,C 180,E1 -4606.16,E2 -4606.16} C_VEL
LIN {X 0,Y 524.3,Z 341.7,A -85,B 0,C 180,E1 -4607.34,E2 -4607.34} C_VEL
LIN {X 0,Y 524.607,Z 332.457,A -85,B 0,C 180,E1 -4608.35,E2 -4608.35} C_VEL
LIN {X 0,Y 524.972,Z 321.48,A -85,B 0,C 180,E1 -4609.35,E2 -4609.35} C_VEL
LIN {X 0,Y 525.307,Z 309.392,A -85,B 0,C 180,E1 -4610.254,E2 -4610.254} C_VEL
LIN {X 0,Y 525.673,Z 297.399,A -85,B 0,C 180,E1 -4610.977,E2 -4610.977} C_VEL
LIN {X 0,Y 526.051,Z 284.108,A -85,B 0,C 180,E1 -4611.607,E2 -4611.607} C_VEL
LIN {X 0,Y 526.306,Z 269.72,A -85,B 0,C 180,E1 -4612.111,E2 -4612.111} C_VEL
LIN {X 0,Y 526.502,Z 255.604,A -85,B 0,C 180,E1 -4612.438,E2 -4612.438} C_VEL
LIN {X 0,Y 527.13,Z 131.548,A -85,B 0,C 180,E1 -4614.168,E2 -4614.168} C_VEL
LIN {X 0,Y 524.907,Z 120.665,A -85,B 0,C 180,E1 -4614.408,E2 -4614.408} C_VEL
LIN {X 0,Y 525.307,Z 104.747,A -85,B 0,C 180,E1 -4617.057,E2 -4617.057} C_VEL
LIN {X 0,Y 525.112,Z 99.529,A -85,B 0,C 180,E1 -4617.952,E2 -4617.952} C_VEL
LIN {X 0,Y 523.892,Z 93.352,A -85,B 0,C 180,E1 -4619.099,E2 -4619.099} C_VEL
LIN {X 0,Y 523.906,Z 93.351,A -85,B 0,C 180,E1 -4621.545,E2 -4621.545} C_VEL
LIN {X 0,Y 523.905,Z 93.351,A -85,B 0,C 180,E1 -4624.292,E2 -4624.292} C_VEL
LIN {X 0,Y 523.873,Z 93.355,A -85,B 0,C 180,E1 -4627.672,E2 -4627.672} C_VEL
LIN {X 0,Y 523.883,Z 93.354,A -85,B 0,C 180,E1 -4630.122,E2 -4630.122} C_VEL
LIN {X 0,Y 523.872,Z 93.353,A -85,B 0,C 180,E1 -4633.172,E2 -4633.172} C_VEL
LIN {X 0,Y 523.919,Z 93.347,A -85,B 0,C 180,E1 -4635.769,E2 -4635.769} C_VEL
LIN {X 0,Y 523.892,Z 93.349,A -85,B 0,C 180,E1 -4638.903,E2 -4638.903} C_VEL
LIN {X 0,Y 523.902,Z 93.348,A -85,B 0,C 180,E1 -4641.897,E2 -4641.897} C_VEL
LIN {X 0,Y 523.919,Z 93.347,A -85,B 0,C 180,E1 -4644.912,E2 -4644.912} C_VEL
LIN {X 0,Y 523.936,Z 93.344,A -85,B 0,C 180,E1 -4647.68,E2 -4647.68} C_VEL
LIN {X 0,Y 523.936,Z 93.344,A -85,B 0,C 180,E1 -4650.68,E2 -4650.68} C_VEL
LIN {X 0,Y 523.903,Z 93.344,A -85,B 0,C 180,E1 -4653.724,E2 -4653.724} C_VEL
LIN {X 0,Y 523.908,Z 93.347,A -85,B 0,C 180,E1 -4656.269,E2 -4656.269} C_VEL
LIN {X 0,Y 523.944,Z 93.348,A -85,B 0,C 180,E1 -4658.766,E2 -4658.766} C_VEL
LIN {X 0,Y 523.938,Z 93.341,A -85,B 0,C 180,E1 -4661.22,E2 -4661.22} C_VEL
LIN {X 0,Y 523.921,Z 93.344,A -85,B 0,C 180,E1 -4663.638,E2 -4663.638} C_VEL
LIN {X 0,Y 523.917,Z 93.346,A -85,B 0,C 180,E1 -4666.027,E2 -4666.027} C_VEL
LIN {X 0,Y 524.014,Z 93.341,A -85,B 0,C 180,E1 -4668.394,E2 -4668.394} C_VEL
LIN {X 0,Y 523.988,Z 93.332,A -85,B 0,C 180,E1 -4671.516,E2 -4671.516} C_VEL
LIN {X 0,Y 524.075,Z 93.326,A -85,B 0,C 180,E1 -4674.613,E2 -4674.613} C_VEL
LIN {X 0,Y 524.111,Z 93.322,A -85,B 0,C 180,E1 -4677.694,E2 -4677.694} C_VEL
LIN {X 0,Y 524.121,Z 93.316,A -85,B 0,C 180,E1 -4680.768,E2 -4680.768} C_VEL
LIN {X 0,Y 524.041,Z 93.329,A -85,B 0,C 180,E1 -4683.075,E2 -4683.075} C_VEL
LIN {X 0,Y 524.012,Z 93.332,A -85,B 0,C 180,E1 -4686.159,E2 -4686.159} C_VEL
LIN {X 0,Y 523.988,Z 93.339,A -85,B 0,C 180,E1 -4689.262,E2 -4689.262} C_VEL
LIN {X 0,Y 524,Z 93.338,A -85,B 0,C 180,E1 -4691.737,E2 -4691.737} C_VEL
LIN {X 0,Y 523.993,Z 93.339,A -85,B 0,C 180,E1 -4695.052,E2 -4695.052} C_VEL
LIN {X 0,Y 523.964,Z 93.339,A -85,B 0,C 180,E1 -4697.969,E2 -4697.969} C_VEL
LIN {X 0,Y 523.973,Z 93.335,A -85,B 0,C 180,E1 -4700.41,E2 -4700.41} C_VEL
LIN {X 0,Y 523.911,Z 93.35,A -85,B 0,C 180,E1 -4702.893,E2 -4702.893} C_VEL
LIN {X 0,Y 523.954,Z 93.342,A -85,B 0,C 180,E1 -4705.419,E2 -4705.419} C_VEL
LIN {X 0,Y 523.969,Z 93.337,A -85,B 0,C 180,E1 -4707.999,E2 -4707.999} C_VEL
LIN {X 0,Y 523.946,Z 93.348,A -85,B 0,C 180,E1 -4710.855,E2 -4710.855} C_VEL
LIN {X 0,Y 523.961,Z 93.339,A -85,B 0,C 180,E1 -4713.735,E2 -4713.735} C_VEL
LIN {X 0,Y 523.904,Z 93.35,A -85,B 0,C 180,E1 -4716.401,E2 -4716.401} C_VEL
LIN {X 0,Y 523.92,Z 93.34,A -85,B 0,C 180,E1 -4719.085,E2 -4719.085} C_VEL
LIN {X 0,Y 523.955,Z 93.344,A -85,B 0,C 180,E1 -4722.119,E2 -4722.119} C_VEL
LIN {X 0,Y 523.946,Z 93.339,A -85,B 0,C 180,E1 -4725.31,E2 -4725.31} C_VEL
LIN {X 0,Y 523.959,Z 93.341,A -85,B 0,C 180,E1 -4728.689,E2 -4728.689} C_VEL
LIN {X 0,Y 523.921,Z 93.343,A -85,B 0,C 180,E1 -4731.08,E2 -4731.08} C_VEL
LIN {X 0,Y 523.901,Z 93.352,A -85,B 0,C 180,E1 -4733.825,E2 -4733.825} C_VEL
LIN {X 0,Y 523.942,Z 93.339,A -85,B 0,C 180,E1 -4736.636,E2 -4736.636} C_VEL
LIN {X 0,Y 523.957,Z 93.343,A -85,B 0,C 180,E1 -4739.356,E2 -4739.356} C_VEL
LIN {X 0,Y 523.98,Z 93.341,A -85,B 0,C 180,E1 -4742.281,E2 -4742.281} C_VEL
LIN {X 0,Y 523.976,Z 93.433,A -85,B 0,C 180,E1 -4744.292,E2 -4744.292} C_VEL
LIN {X 0,Y 525.841,Z 102.309,A -85,B 0,C 180,E1 -4745.733,E2 -4745.733} C_VEL
LIN {X 0,Y 525.664,Z 113.651,A -85,B 0,C 180,E1 -4747.42,E2 -4747.42} C_VEL
LIN {X 0,Y 525.065,Z 134.476,A -85,B 0,C 180,E1 -4750.45,E2 -4750.45} C_VEL
LIN {X 0,Y 524.886,Z 142.588,A -85,B 0,C 180,E1 -4751.618,E2 -4751.618} C_VEL
LIN {X 0,Y 527.164,Z 155.846,A -85,B 0,C 180,E1 -4751.897,E2 -4751.897} C_VEL
LIN {X 0,Y 526.413,Z 280.899,A -85,B 0,C 180,E1 -4753.643,E2 -4753.643} C_VEL
LIN {X 0,Y 526.176,Z 295.3,A -85,B 0,C 180,E1 -4754.005,E2 -4754.005} C_VEL
LIN {X 0,Y 525.907,Z 308.801,A -85,B 0,C 180,E1 -4754.498,E2 -4754.498} C_VEL
LIN {X 0,Y 525.563,Z 321.004,A -85,B 0,C 180,E1 -4755.083,E2 -4755.083} C_VEL
LIN {X 0,Y 525.143,Z 333.844,A -85,B 0,C 180,E1 -4755.863,E2 -4755.863} C_VEL
LIN {X 0,Y 524.785,Z 345.522,A -85,B 0,C 180,E1 -4756.742,E2 -4756.742} C_VEL
LIN {X 0,Y 524.44,Z 356.39,A -85,B 0,C 180,E1 -4757.734,E2 -4757.734} C_VEL
LIN {X 0,Y 524.18,Z 366.011,A -85,B 0,C 180,E1 -4758.79,E2 -4758.79} C_VEL
LIN {X 0,Y 523.852,Z 374.903,A -85,B 0,C 180,E1 -4759.956,E2 -4759.956} C_VEL
LIN {X 0,Y 523.708,Z 382.306,A -85,B 0,C 180,E1 -4761.122,E2 -4761.122} C_VEL
LIN {X 0,Y 523.561,Z 388.477,A -85,B 0,C 180,E1 -4762.286,E2 -4762.286} C_VEL
LIN {X 0,Y 523.437,Z 395.031,A -85,B 0,C 180,E1 -4763.834,E2 -4763.834} C_VEL
LIN {X 0,Y 523.375,Z 398.867,A -85,B 0,C 180,E1 -4764.993,E2 -4764.993} C_VEL
LIN {X 0,Y 523.418,Z 401.823,A -85,B 0,C 180,E1 -4766.15,E2 -4766.15} C_VEL
LIN {X 0,Y 523.333,Z 404.527,A -85,B 0,C 180,E1 -4767.691,E2 -4767.691} C_VEL
LIN {X 0,Y 523.246,Z 405.867,A -85,B 0,C 180,E1 -4769.23,E2 -4769.23} C_VEL
LIN {X 0,Y 523.246,Z 405.868,A -85,B 0,C 180,E1 -4770.769,E2 -4770.769} C_VEL
LIN {X 0,Y 523.333,Z 404.533,A -85,B 0,C 180,E1 -4772.309,E2 -4772.309} C_VEL
LIN {X 0,Y 523.418,Z 401.832,A -85,B 0,C 180,E1 -4773.849,E2 -4773.849} C_VEL
LIN {X 0,Y 523.443,Z 397.688,A -85,B 0,C 180,E1 -4775.393,E2 -4775.393} C_VEL
LIN {X 0,Y 523.493,Z 391.979,A -85,B 0,C 180,E1 -4776.94,E2 -4776.94} C_VEL
LIN {X 0,Y 523.619,Z 385.544,A -85,B 0,C 180,E1 -4778.296,E2 -4778.296} C_VEL
LIN {X 0,Y 523.822,Z 377.55,A -85,B 0,C 180,E1 -4779.655,E2 -4779.655} C_VEL
LIN {X 0,Y 524.078,Z 369.189,A -85,B 0,C 180,E1 -4780.821,E2 -4780.821} C_VEL
LIN {X 0,Y 524.417,Z 358.514,A -85,B 0,C 180,E1 -4782.055,E2 -4782.055} C_VEL
LIN {X 0,Y 524.724,Z 347.897,A -85,B 0,C 180,E1 -4783.063,E2 -4783.063} C_VEL
LIN {X 0,Y 525.092,Z 335.302,A -85,B 0,C 180,E1 -4784.039,E2 -4784.039} C_VEL
LIN {X 0,Y 525.503,Z 322.802,A -85,B 0,C 180,E1 -4784.819,E2 -4784.819} C_VEL
LIN {X 0,Y 525.873,Z 309.953,A -85,B 0,C 180,E1 -4785.453,E2 -4785.453} C_VEL
LIN {X 0,Y 526.167,Z 295.79,A -85,B 0,C 180,E1 -4785.98,E2 -4785.98} C_VEL
LIN {X 0,Y 526.42,Z 282.077,A -85,B 0,C 180,E1 -4786.331,E2 -4786.331} C_VEL
LIN {X 0,Y 526.604,Z 255.744,A -85,B 0,C 180,E1 -4786.724,E2 -4786.724} C_VEL
LIN {X 0,Y 527.065,Z 154.899,A -85,B 0,C 180,E1 -4788.12,E2 -4788.12} C_VEL
LIN {X 0,Y 524.89,Z 142.612,A -85,B 0,C 180,E1 -4788.383,E2 -4788.383} C_VEL
LIN {X 0,Y 525.376,Z 123.293,A -85,B 0,C 180,E1 -4791.173,E2 -4791.173} C_VEL
LIN {X 0,Y 525.948,Z 103.586,A -85,B 0,C 180,E1 -4794.051,E2 -4794.051} C_VEL
LIN {X 0,Y 523.991,Z 93.342,A -85,B 0,C 180,E1 -4795.685,E2 -4795.685} C_VEL
LIN {X 0,Y 523.97,Z 93.343,A -85,B 0,C 180,E1 -4797.999,E2 -4797.999} C_VEL
LIN {X 0,Y 523.945,Z 93.344,A -85,B 0,C 180,E1 -4800.854,E2 -4800.854} C_VEL
LIN {X 0,Y 523.959,Z 93.341,A -85,B 0,C 180,E1 -4803.734,E2 -4803.734} C_VEL
LIN {X 0,Y 523.903,Z 93.35,A -85,B 0,C 180,E1 -4806.401,E2 -4806.401} C_VEL
LIN {X 0,Y 523.923,Z 93.343,A -85,B 0,C 180,E1 -4809.084,E2 -4809.084} C_VEL
LIN {X 0,Y 523.955,Z 93.344,A -85,B 0,C 180,E1 -4812.118,E2 -4812.118} C_VEL
LIN {X 0,Y 523.956,Z 93.341,A -85,B 0,C 180,E1 -4815.308,E2 -4815.308} C_VEL
LIN {X 0,Y 523.958,Z 93.338,A -85,B 0,C 180,E1 -4818.689,E2 -4818.689} C_VEL
LIN {X 0,Y 523.916,Z 93.346,A -85,B 0,C 180,E1 -4821.08,E2 -4821.08} C_VEL
LIN {X 0,Y 523.899,Z 93.35,A -85,B 0,C 180,E1 -4823.825,E2 -4823.825} C_VEL
LIN {X 0,Y 523.941,Z 93.341,A -85,B 0,C 180,E1 -4826.636,E2 -4826.636} C_VEL
LIN {X 0,Y 523.955,Z 93.348,A -85,B 0,C 180,E1 -4829.356,E2 -4829.356} C_VEL
LIN {X 0,Y 523.976,Z 93.336,A -85,B 0,C 180,E1 -4832.281,E2 -4832.281} C_VEL
LIN {X 0,Y 523.952,Z 93.341,A -85,B 0,C 180,E1 -4834.581,E2 -4834.581} C_VEL
LIN {X 0,Y 523.91,Z 93.353,A -85,B 0,C 180,E1 -4837.106,E2 -4837.106} C_VEL
LIN {X 0,Y 523.978,Z 93.336,A -85,B 0,C 180,E1 -4839.866,E2 -4839.866} C_VEL
LIN {X 0,Y 523.965,Z 93.346,A -85,B 0,C 180,E1 -4842.837,E2 -4842.837} C_VEL
LIN {X 0,Y 523.976,Z 93.339,A -85,B 0,C 180,E1 -4845.236,E2 -4845.236} C_VEL
LIN {X 0,Y 524.012,Z 93.336,A -85,B 0,C 180,E1 -4848.394,E2 -4848.394} C_VEL
LIN {X 0,Y 524.002,Z 93.333,A -85,B 0,C 180,E1 -4851.516,E2 -4851.516} C_VEL
LIN {X 0,Y 524.08,Z 93.33,A -85,B 0,C 180,E1 -4854.614,E2 -4854.614} C_VEL
LIN {X 0,Y 524.11,Z 93.32,A -85,B 0,C 180,E1 -4857.695,E2 -4857.695} C_VEL
LIN {X 0,Y 524.121,Z 93.321,A -85,B 0,C 180,E1 -4860.768,E2 -4860.768} C_VEL
LIN {X 0,Y 524.07,Z 93.325,A -85,B 0,C 180,E1 -4863.075,E2 -4863.075} C_VEL
LIN {X 0,Y 524.025,Z 93.338,A -85,B 0,C 180,E1 -4866.159,E2 -4866.159} C_VEL
LIN {X 0,Y 524.003,Z 93.336,A -85,B 0,C 180,E1 -4868.484,E2 -4868.484} C_VEL
LIN {X 0,Y 524.002,Z 93.339,A -85,B 0,C 180,E1 -4871.74,E2 -4871.74} C_VEL
LIN {X 0,Y 523.993,Z 93.335,A -85,B 0,C 180,E1 -4875.053,E2 -4875.053} C_VEL
LIN {X 0,Y 523.944,Z 93.345,A -85,B 0,C 180,E1 -4877.97,E2 -4877.97} C_VEL
LIN {X 0,Y 523.972,Z 93.337,A -85,B 0,C 180,E1 -4880.41,E2 -4880.41} C_VEL
LIN {X 0,Y 523.91,Z 93.346,A -85,B 0,C 180,E1 -4882.894,E2 -4882.894} C_VEL
LIN {X 0,Y 523.984,Z 93.337,A -85,B 0,C 180,E1 -4886.02,E2 -4886.02} C_VEL
LIN {X 0,Y 523.93,Z 93.345,A -85,B 0,C 180,E1 -4888.876,E2 -4888.876} C_VEL
LIN {X 0,Y 523.919,Z 93.348,A -85,B 0,C 180,E1 -4891.545,E2 -4891.545} C_VEL
LIN {X 0,Y 523.92,Z 93.343,A -85,B 0,C 180,E1 -4894.291,E2 -4894.291} C_VEL
LIN {X 0,Y 523.907,Z 93.353,A -85,B 0,C 180,E1 -4897.133,E2 -4897.133} C_VEL
LIN {X 0,Y 523.938,Z 93.341,A -85,B 0,C 180,E1 -4900.13,E2 -4900.13} C_VEL
LIN {X 0,Y 523.936,Z 93.344,A -85,B 0,C 180,E1 -4902.459,E2 -4902.459} C_VEL
LIN {X 0,Y 523.946,Z 93.342,A -85,B 0,C 180,E1 -4905.31,E2 -4905.31} C_VEL
LIN {X 0,Y 523.901,Z 93.352,A -85,B 0,C 180,E1 -4906.898,E2 -4906.898} C_VEL
LIN {X 0,Y 523.24,Z 93.43,A -85,B 0,C 180,E1 -4907.539,E2 -4907.539} C_VEL
LIN {X 0,Y 520.406,Z 93.788,A -85,B 0,C 180,E1 -4908.581,E2 -4908.581} C_VEL
LIN {X 0,Y 518.007,Z 94.086,A -85,B 0,C 180,E1 -4909.42,E2 -4909.42} C_VEL
LIN {X 0,Y 516.97,Z 94.213,A -85,B 0,C 180,E1 -4910.068,E2 -4910.068} C_VEL
LIN {X 0,Y 516.882,Z 94.224,A -85,B 0,C 180,E1 -4910.287,E2 -4910.287} C_VEL
LIN {X 0,Y 516.854,Z 94.224,A -85,B 0,C 180,E1 -4913.347,E2 -4913.347} C_VEL
LIN {X 0,Y 516.908,Z 94.221,A -85,B 0,C 180,E1 -4916.121,E2 -4916.121} C_VEL
LIN {X 0,Y 516.893,Z 94.22,A -85,B 0,C 180,E1 -4918.936,E2 -4918.936} C_VEL
LIN {X 0,Y 516.863,Z 94.223,A -85,B 0,C 180,E1 -4921.582,E2 -4921.582} C_VEL
